// TIA Portal project "Tester_Forma_W1" (V16)
// Program sterowania formą wtryskarki do zalewania gumą końcuwek rur.

(* hardware
DEVICE "Tester_Forma"  S7-1200 Station
   slot 0: "Rack_0"  S7-1200 Rack  Rack  V1.0
   slot 1: "PLC_1"  CPU 1214C AC/DC/Rly  6ES7 214-1BG40-0XB0  V4.4
   slot 2: "DI 16x24VDC/DQ 16xRelay_1"  SM 1223 DI16/DQ16 x relay  6ES7 223-1PL32-0XB0  V2.0
   slot 3: "DQ 8x24VDC _1"  SM 1222 DQ8 x 24VDC  6ES7 222-1BF32-0XB0  V2.0
DEVICE "HMI_1"  KTP400 Basic PN
   slot 0: "HMI_1"  KTP400 Basic PN  6AV2 123-2DB03-0AX0  15.1.0.0
   slot 1: "HMI_RT_1"  KTP400 Basic PN  6AV2 123-2DB03-0AX0  15.1.0.0
   slot 5: "HMI_1.IE_CP_1"  PROFINET Interface  15.0.1.0
      slot 1: "PROFINET Interface_1"  PROFINET Interface
         slot 1: "Port_1"  Port
*)

// ===== PLC "PLC_1"  CPU 1214C AC/DC/Rly =====

VAR_GLOBAL   // PLC tag table "Default tag table"
   "System_Byte" AT %MB1 : Byte;
   "FirstScan" AT %M1.0 : Bool;
   "DiagStatusUpdate" AT %M1.1 : Bool;
   "AlwaysTRUE" AT %M1.2 : Bool;
   "AlwaysFALSE" AT %M1.3 : Bool;
   "Clock_Byte" AT %MB0 : Byte;
   "Clock_10Hz" AT %M0.0 : Bool;
   "Clock_5Hz" AT %M0.1 : Bool;
   "Clock_2.5Hz" AT %M0.2 : Bool;
   "Clock_2Hz" AT %M0.3 : Bool;
   "Clock_1.25Hz" AT %M0.4 : Bool;
   "Clock_1Hz" AT %M0.5 : Bool;
   "Clock_0.625Hz" AT %M0.6 : Bool;
   "Clock_0.5Hz" AT %M0.7 : Bool;
END_VAR

VAR_GLOBAL   // PLC tag table "InputsPLC"
   "diSE_OpenGripper1" AT %I0.0 : Bool;
   "diSE_OpenGripper2" AT %I0.1 : Bool;
   "diSE_OpenGripper3" AT %I0.2 : Bool;
   "diSE_OpenGripper4" AT %I0.3 : Bool;
   "diSE_OpenGripper5" AT %I0.4 : Bool;
   "diSE_OpenGripper6" AT %I0.5 : Bool;
   "diSE_OpenGripper7" AT %I0.6 : Bool;
   "diSE_OpenGripper8" AT %I0.7 : Bool;
   "diSE_PresencePin1" AT %I1.0 : Bool;
   "diSE_PresencePin2" AT %I1.1 : Bool;
   "diSE_PresencePin3" AT %I1.2 : Bool;
   "diSE_PresencePin4" AT %I1.3 : Bool;
   "diSE_PresencePin5" AT %I1.4 : Bool;
   "diSE_PresencePin6" AT %I1.5 : Bool;
   "diSE_PresencePin7" AT %I8.0 : Bool;
   "diSE_PresencePin8" AT %I8.1 : Bool;
   "diSE_LeftActuatorGrippersUpPosition" AT %I8.2 : Bool;
   "diSE_LeftActuatorGrippersDownPosition" AT %I8.3 : Bool;
   "diSE_LeftActuatorTablePinsDownPosition" AT %I8.4 : Bool;
   "diSE_LeftActuatorTablePinsUpPositon" AT %I8.5 : Bool;
   "diSE_RightActuatorTablePinsDownPositon" AT %I8.6 : Bool;
   "diSE_RightActuatorTablePinsUpPosition" AT %I8.7 : Bool;
   "diSE_RightActuatorGripperUpPosition" AT %I9.0 : Bool;
   "diSE_RightActuatorGripperDownPositon" AT %I9.1 : Bool;
   "diPressOpenedUp" AT %I9.4 : Bool;
   "diPressClosedDown" AT %I9.6 : Bool;
   "diPreventaOK" AT %I9.2 : Bool;
   "diBT_Reset" AT %I9.3 : Bool;
   "diBT_StartCycle2" AT %I9.5 : Bool;
   "diPressInjectionEnd" AT %I9.7 : Bool;
END_VAR

VAR_GLOBAL   // PLC tag table "OutputsPLC"
   "dqPermitToClosePress" AT %Q0.0 : Bool;
   "dqPressInterface1" AT %Q0.1 : Bool;
   "dqPressInterface2" AT %Q0.2 : Bool;
   "dqPressInterface3" AT %Q0.3 : Bool;
   "dqReserveQ0_4" AT %Q0.4 : Bool;
   "dqReserveQ0_5" AT %Q0.5 : Bool;
   "dqLED_RedFault" AT %Q0.6 : Bool;
   "dqBuzzer" AT %Q0.7 : Bool;
   "dqReserveQ1_0" AT %Q1.0 : Bool;
   "dqReserveQ1_1" AT %Q1.1 : Bool;
   "dqTablePinsUp" AT %Q8.0 : Bool;
   "dqTablePinsDown" AT %Q8.1 : Bool;
   "dqGrippresDown" AT %Q8.2 : Bool;
   "dqGrippersUp" AT %Q8.3 : Bool;
   "dqOpeningGripper1" AT %Q8.4 : Bool;
   "dqClosingGripper1" AT %Q8.5 : Bool;
   "dqOpeningGripper2" AT %Q8.6 : Bool;
   "dqClosingGripper2" AT %Q8.7 : Bool;
   "dqOpeningGripper3" AT %Q9.0 : Bool;
   "dqClosingGripper3" AT %Q9.1 : Bool;
   "dqOpeningGripper4" AT %Q9.2 : Bool;
   "dqClosingGripper4" AT %Q9.3 : Bool;
   "dqOpeningGripper5" AT %Q9.4 : Bool;
   "dqClosingGripper5" AT %Q9.5 : Bool;
   "dqOpeningGripper6" AT %Q9.6 : Bool;
   "dqClosingGripper6" AT %Q9.7 : Bool;
   "dqOpeningGripper7" AT %Q12.0 : Bool;
   "dqClosingGripper7" AT %Q12.1 : Bool;
   "dqOpeningGripper8" AT %Q12.2 : Bool;
   "dqClosingGripper8" AT %Q12.3 : Bool;
   "dqReserveq12_4" AT %Q12.4 : Bool;
   "dqReserveq12_5" AT %Q12.5 : Bool;
   "dqReserveq12_6" AT %Q12.6 : Bool;
   "dqReserveq12_7" AT %Q12.7 : Bool;
END_VAR

DATA_BLOCK "Variable"   // DB1
{ S7_Optimized_Access := 'TRUE' }
VERSION : 0.1
   VAR
      FirstScanDone : Bool;
      SetMachineInitialStatus : Bool;
   END_VAR
   VAR RETAIN
      M_EvTableGrippres : Bool;
      M_EvTablePins : Bool;
   END_VAR
   VAR
      OutBuzzerPinActivatedByTube1 : Bool;
      OutBuzzerPinActivatedByTube2 : Bool;
      OutBuzzerPinActivatedByTube3 : Bool;
      OutBuzzerPinActivatedByTube4 : Bool;
      OutBuzzerPinActivatedByTube5 : Bool;
      OutBuzzerPinActivatedByTube6 : Bool;
      OutBuzzerPinActivatedByTube7 : Bool;
      OutBuzzerPinActivatedByTube8 : Bool;
   END_VAR
   VAR RETAIN
      BuzzerDurationSignal : Time := T#100ms;
   END_VAR
   VAR
      SignalBuzzerPinPresent : Bool;
      M_PinsNotActivated : Bool;
      M_PinsActivated : Bool;
      M_GrippersOpened : Bool;
      M_GrippersClosed : Bool;
      M_PinsTableUpPosition : Bool;
      M_PinsTableDownPosition : Bool;
      M_GrippersTableUpPositon : Bool;
      M_GrippersTableDownPositon : Bool;
      M_EvGripperOutput1 : Bool;
      M_EvGripperOutput2 : Bool;
      M_EvGripperOutput3 : Bool;
      M_EvGripperOutput4 : Bool;
      M_EvGripperOutput5 : Bool;
      M_EvGripperOutput6 : Bool;
      M_EvGripperOutput7 : Bool;
      M_EvGripperOutput8 : Bool;
      M_ReadyForFirstCycle : Bool;
      M_PreparePositionForFirstStart : Bool;
      M_StartCycleButtons : Bool;
      M_EvGrippresInitial : Bool;
      M_EvTablePinsInitial : Bool := false;
      M_EvGripperOutputInitial : Bool;
      M_AutomaticModePermissionToCloseGrippers : Bool;
   END_VAR
BEGIN
END_DATA_BLOCK

DATA_BLOCK "HMI"   // DB8
{ S7_Optimized_Access := 'FALSE' }
VERSION : 0.1
   VAR
      Auto : Bool := false;
      Manu : Bool;
      OpenInAutoGripper1 : Bool;
      OpenInAutoGripper2 : Bool;
      OpenInAutoGripper3 : Bool;
      OpenInAutoGripper4 : Bool;
      OpenInAutoGripper5 : Bool;
      OpenInAutoGripper6 : Bool;
      OpenInAutoGripper7 : Bool;
      OpenInAutoGripper8 : Bool;
      OpenInManuGripper1 : Bool;
      OpenInManuGripper2 : Bool;
      OpenInManuGripper3 : Bool;
      OpenInManuGripper4 : Bool;
      OpenInManuGripper5 : Bool;
      OpenInManuGripper6 : Bool;
      OpenInManuGripper7 : Bool;
      OpenInManuGripper8 : Bool;
      CloseInManuGripper1 : Bool;
      CloseInManuGripper2 : Bool;
      CloseInManuGripper3 : Bool;
      CloseInManuGripper4 : Bool;
      CloseInManuGripper5 : Bool;
      CloseInManuGripper6 : Bool;
      CloseInManuGripper7 : Bool;
      CloseInManuGripper8 : Bool;
      TableGrippersUP : Bool;
      TableGripperDown : Bool;
      TablePinsUp : Bool;
      TablePinsDown : Bool;
      OpenManuAllGrippers : Bool;
   END_VAR
BEGIN
END_DATA_BLOCK

DATA_BLOCK "MemoryEdge"   // DB9
{ S7_Optimized_Access := 'TRUE' }
VERSION : 0.1
   VAR
      Memory1 : Bool;
      Memory2 : Bool;
      Memory3 : Bool;
      Memory4 : Bool;
      Memory5 : Bool;
      Memory6 : Bool;
      Memory7 : Bool;
      Memory8 : Bool;
      Memory9 : Bool;
      Memory10 : Bool;
      Memory11 : Bool;
      Memory12 : Bool;
      Memory13 : Bool;
      Memory14 : Bool;
   END_VAR
BEGIN
END_DATA_BLOCK

DATA_BLOCK "Outputs_DB"   // DB16
{ S7_Optimized_Access := 'TRUE' }
VERSION : 0.1
// stored: InstanceOfName Outputs
"Outputs"
BEGIN
END_DATA_BLOCK

DATA_BLOCK "AlarmsBlock"   // DB17
{ S7_Optimized_Access := 'FALSE' }
VERSION : 0.1
   VAR
      AlarmOccurred : Bool;
      AlarmLeftActuatorGrippers : Bool;
      AlarmRightActuatorGrippers : Bool;
      AlarmLeftActuatorPins : Bool;
      AlarmRightActuatorPins : Bool;
      M_AlarmGripper1 : Bool;
      M_AlarmGripper2 : Bool;
      M_AlarmGripper3 : Bool;
      M_AlarmGripper4 : Bool;
      M_AlarmGripper5 : Bool;
      M_AlarmGripper6 : Bool;
      M_AlarmGripper7 : Bool;
      M_AlarmGripper8 : Bool;
   END_VAR
BEGIN
END_DATA_BLOCK

// folder: GripperError

DATA_BLOCK "Gripper6_Error"   // DB6
{ S7_Optimized_Access := 'TRUE' }
VERSION : 0.1
// stored: InstanceOfName GripperError
"GripperError"
BEGIN
END_DATA_BLOCK

DATA_BLOCK "Gripper1_Error"   // DB7
{ S7_Optimized_Access := 'TRUE' }
VERSION : 0.1
// stored: InstanceOfName GripperError
"GripperError"
BEGIN
END_DATA_BLOCK

DATA_BLOCK "Gripper2_Error"   // DB10
{ S7_Optimized_Access := 'TRUE' }
VERSION : 0.1
// stored: InstanceOfName GripperError
"GripperError"
BEGIN
END_DATA_BLOCK

DATA_BLOCK "Gripper3_Error"   // DB11
{ S7_Optimized_Access := 'TRUE' }
VERSION : 0.1
// stored: InstanceOfName GripperError
"GripperError"
BEGIN
END_DATA_BLOCK

DATA_BLOCK "Gripper4_Error"   // DB12
{ S7_Optimized_Access := 'TRUE' }
VERSION : 0.1
// stored: InstanceOfName GripperError
"GripperError"
BEGIN
END_DATA_BLOCK

DATA_BLOCK "Gripper5_Error"   // DB13
{ S7_Optimized_Access := 'TRUE' }
VERSION : 0.1
// stored: InstanceOfName GripperError
"GripperError"
BEGIN
END_DATA_BLOCK

DATA_BLOCK "Gripper7_Error"   // DB14
{ S7_Optimized_Access := 'TRUE' }
VERSION : 0.1
// stored: InstanceOfName GripperError
"GripperError"
BEGIN
END_DATA_BLOCK

DATA_BLOCK "Gripper8_Error"   // DB15
{ S7_Optimized_Access := 'TRUE' }
VERSION : 0.1
// stored: InstanceOfName GripperError
"GripperError"
BEGIN
END_DATA_BLOCK

// folder: GripperOpenClose

DATA_BLOCK "GripperOpenCloseAutoManu_DB1"   // DB18
{ S7_Optimized_Access := 'TRUE' }
VERSION : 0.1
// stored: InstanceOfName GripperOpenCloseAutoManu
"GripperOpenCloseAutoManu"
BEGIN
END_DATA_BLOCK

DATA_BLOCK "GripperOpenCloseAutoManu_DB"   // DB19
{ S7_Optimized_Access := 'TRUE' }
VERSION : 0.1
// stored: InstanceOfName GripperOpenCloseAutoManu
"GripperOpenCloseAutoManu"
BEGIN
END_DATA_BLOCK

DATA_BLOCK "GripperOpenCloseAutoManu_DB_1"   // DB20
{ S7_Optimized_Access := 'TRUE' }
VERSION : 0.1
// stored: InstanceOfName GripperOpenCloseAutoManu
"GripperOpenCloseAutoManu"
BEGIN
END_DATA_BLOCK

DATA_BLOCK "GripperOpenCloseAutoManu_DB_2"   // DB21
{ S7_Optimized_Access := 'TRUE' }
VERSION : 0.1
// stored: InstanceOfName GripperOpenCloseAutoManu
"GripperOpenCloseAutoManu"
BEGIN
END_DATA_BLOCK

DATA_BLOCK "GripperOpenCloseAutoManu_DB_3"   // DB22
{ S7_Optimized_Access := 'TRUE' }
VERSION : 0.1
// stored: InstanceOfName GripperOpenCloseAutoManu
"GripperOpenCloseAutoManu"
BEGIN
END_DATA_BLOCK

DATA_BLOCK "GripperOpenCloseAutoManu_DB_4"   // DB23
{ S7_Optimized_Access := 'TRUE' }
VERSION : 0.1
// stored: InstanceOfName GripperOpenCloseAutoManu
"GripperOpenCloseAutoManu"
BEGIN
END_DATA_BLOCK

DATA_BLOCK "GripperOpenCloseAutoManu_DB_5"   // DB24
{ S7_Optimized_Access := 'TRUE' }
VERSION : 0.1
// stored: InstanceOfName GripperOpenCloseAutoManu
"GripperOpenCloseAutoManu"
BEGIN
END_DATA_BLOCK

DATA_BLOCK "GripperOpenCloseAutoManu_DB_6"   // DB25
{ S7_Optimized_Access := 'TRUE' }
VERSION : 0.1
// stored: InstanceOfName GripperOpenCloseAutoManu
"GripperOpenCloseAutoManu"
BEGIN
END_DATA_BLOCK

// folder: System blocks/Program resources

DATA_BLOCK "TimeToAlarmLeftActuatoGrippers"   // DB2
{ S7_Optimized_Access := 'TRUE' }
AUTHOR : Simatic
FAMILY : IEC
NAME : IEC_TMR
VERSION : 1.0
// stored: InstanceOfName IEC_TIMER
"IEC_TIMER"
BEGIN
END_DATA_BLOCK

DATA_BLOCK "TimeToAlarmRightActuatoGrippers"   // DB3
{ S7_Optimized_Access := 'TRUE' }
AUTHOR : Simatic
FAMILY : IEC
NAME : IEC_TMR
VERSION : 1.0
// stored: InstanceOfName IEC_TIMER
"IEC_TIMER"
BEGIN
END_DATA_BLOCK

DATA_BLOCK "TimeToAlarmLeftActuatoPins"   // DB4
{ S7_Optimized_Access := 'TRUE' }
AUTHOR : Simatic
FAMILY : IEC
NAME : IEC_TMR
VERSION : 1.0
// stored: InstanceOfName IEC_TIMER
"IEC_TIMER"
BEGIN
END_DATA_BLOCK

DATA_BLOCK "TimeToAlarmRightActuatorPins"   // DB5
{ S7_Optimized_Access := 'TRUE' }
AUTHOR : Simatic
FAMILY : IEC
NAME : IEC_TMR
VERSION : 1.0
// stored: InstanceOfName IEC_TIMER
"IEC_TIMER"
BEGIN
END_DATA_BLOCK

// folder: (top level)

FUNCTION_BLOCK "Outputs"   // FB2, LAD
{ S7_Optimized_Access := 'TRUE' }
VERSION : 0.1
   VAR
      ElectricValve_Grippers : "ElectricValve";
      ElectricValve_TablePins : "ElectricValve";
      ElectricValve_Gripper1 : "ElectricValve";
      ElectricValve_Gripper2 : "ElectricValve";
      ElectricValve_Gripper3 : "ElectricValve";
      ElectricValve_Gripper4 : "ElectricValve";
      ElectricValve_Gripper5 : "ElectricValve";
      ElectricValve_Gripper6 : "ElectricValve";
      ElectricValve_Gripper7 : "ElectricValve";
      ElectricValve_Gripper8 : "ElectricValve";
      Gripper1_Present_Signal : "Buzzer";
      Gripper2_Present_Signal : "Buzzer";
      Gripper3_Present_Signal : "Buzzer";
      Gripper4_Present_Signal : "Buzzer";
      Gripper5_Present_Signal : "Buzzer";
      Gripper6_Present_Signal : "Buzzer";
      Gripper7_Present_Signal : "Buzzer";
      Gripper8_Present_Signal : "Buzzer";
   END_VAR
BEGIN

REGION Network 1: Actuator of Grippers control.
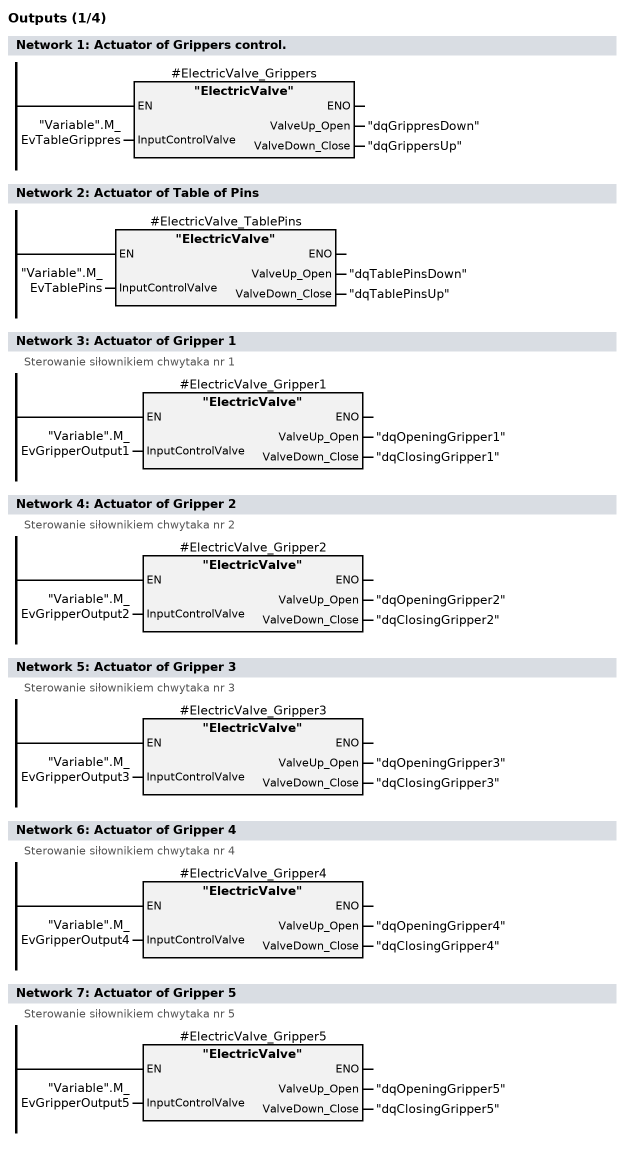
   RUNG wire#powerrail
      #ElectricValve_Grippers(InputControlValve := "Variable".M_EvTableGrippres, ValveUp_Open => "dqGrippresDown", ValveDown_Close => "dqGrippersUp")
   END_RUNG
   // the same network as SCL:
   #ElectricValve_Grippers(InputControlValve := "Variable".M_EvTableGrippres,   // "ElectricValve"
                           ValveUp_Open => "dqGrippresDown",
                           ValveDown_Close => "dqGrippersUp");
END_REGION

REGION Network 2: Actuator of Table of Pins
   RUNG wire#powerrail
      #ElectricValve_TablePins(InputControlValve := "Variable".M_EvTablePins, ValveUp_Open => "dqTablePinsDown", ValveDown_Close => "dqTablePinsUp")
   END_RUNG
   // the same network as SCL:
   #ElectricValve_TablePins(InputControlValve := "Variable".M_EvTablePins,   // "ElectricValve"
                           ValveUp_Open => "dqTablePinsDown",
                           ValveDown_Close => "dqTablePinsUp");
END_REGION

REGION Network 3: Actuator of Gripper 1
   // Sterowanie siłownikiem chwytaka nr 1
   RUNG wire#powerrail
      #ElectricValve_Gripper1(InputControlValve := "Variable".M_EvGripperOutput1, ValveUp_Open => "dqOpeningGripper1", ValveDown_Close => "dqClosingGripper1")
   END_RUNG
   // the same network as SCL:
   #ElectricValve_Gripper1(InputControlValve := "Variable".M_EvGripperOutput1,   // "ElectricValve"
                           ValveUp_Open => "dqOpeningGripper1",
                           ValveDown_Close => "dqClosingGripper1");
END_REGION

REGION Network 4: Actuator of Gripper 2
   // Sterowanie siłownikiem chwytaka nr 2
   RUNG wire#powerrail
      #ElectricValve_Gripper2(InputControlValve := "Variable".M_EvGripperOutput2, ValveUp_Open => "dqOpeningGripper2", ValveDown_Close => "dqClosingGripper2")
   END_RUNG
   // the same network as SCL:
   #ElectricValve_Gripper2(InputControlValve := "Variable".M_EvGripperOutput2,   // "ElectricValve"
                           ValveUp_Open => "dqOpeningGripper2",
                           ValveDown_Close => "dqClosingGripper2");
END_REGION

REGION Network 5: Actuator of Gripper 3
   // Sterowanie siłownikiem chwytaka nr 3
   RUNG wire#powerrail
      #ElectricValve_Gripper3(InputControlValve := "Variable".M_EvGripperOutput3, ValveUp_Open => "dqOpeningGripper3", ValveDown_Close => "dqClosingGripper3")
   END_RUNG
   // the same network as SCL:
   #ElectricValve_Gripper3(InputControlValve := "Variable".M_EvGripperOutput3,   // "ElectricValve"
                           ValveUp_Open => "dqOpeningGripper3",
                           ValveDown_Close => "dqClosingGripper3");
END_REGION

REGION Network 6: Actuator of Gripper 4
   // Sterowanie siłownikiem chwytaka nr 4
   RUNG wire#powerrail
      #ElectricValve_Gripper4(InputControlValve := "Variable".M_EvGripperOutput4, ValveUp_Open => "dqOpeningGripper4", ValveDown_Close => "dqClosingGripper4")
   END_RUNG
   // the same network as SCL:
   #ElectricValve_Gripper4(InputControlValve := "Variable".M_EvGripperOutput4,   // "ElectricValve"
                           ValveUp_Open => "dqOpeningGripper4",
                           ValveDown_Close => "dqClosingGripper4");
END_REGION

REGION Network 7: Actuator of Gripper 5
   // Sterowanie siłownikiem chwytaka nr 5
   RUNG wire#powerrail
      #ElectricValve_Gripper5(InputControlValve := "Variable".M_EvGripperOutput5, ValveUp_Open => "dqOpeningGripper5", ValveDown_Close => "dqClosingGripper5")
   END_RUNG
   // the same network as SCL:
   #ElectricValve_Gripper5(InputControlValve := "Variable".M_EvGripperOutput5,   // "ElectricValve"
                           ValveUp_Open => "dqOpeningGripper5",
                           ValveDown_Close => "dqClosingGripper5");
END_REGION

REGION Network 8: Actuator of Gripper 6
   // Sterowanie siłownikiem chwytaka nr  6
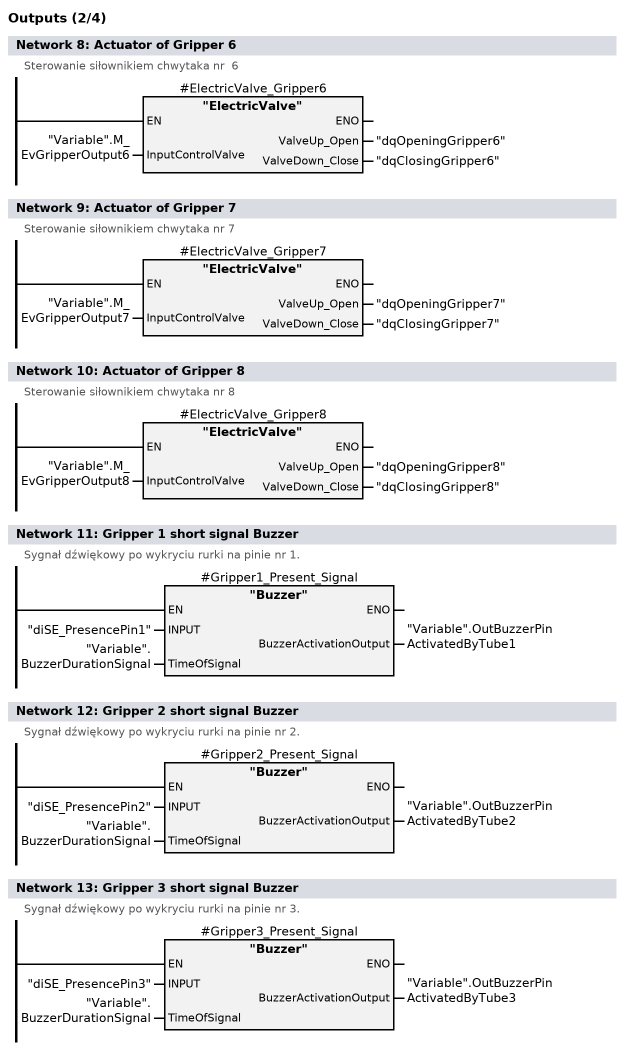
   RUNG wire#powerrail
      #ElectricValve_Gripper6(InputControlValve := "Variable".M_EvGripperOutput6, ValveUp_Open => "dqOpeningGripper6", ValveDown_Close => "dqClosingGripper6")
   END_RUNG
   // the same network as SCL:
   #ElectricValve_Gripper6(InputControlValve := "Variable".M_EvGripperOutput6,   // "ElectricValve"
                           ValveUp_Open => "dqOpeningGripper6",
                           ValveDown_Close => "dqClosingGripper6");
END_REGION

REGION Network 9: Actuator of Gripper 7
   // Sterowanie siłownikiem chwytaka nr 7
   RUNG wire#powerrail
      #ElectricValve_Gripper7(InputControlValve := "Variable".M_EvGripperOutput7, ValveUp_Open => "dqOpeningGripper7", ValveDown_Close => "dqClosingGripper7")
   END_RUNG
   // the same network as SCL:
   #ElectricValve_Gripper7(InputControlValve := "Variable".M_EvGripperOutput7,   // "ElectricValve"
                           ValveUp_Open => "dqOpeningGripper7",
                           ValveDown_Close => "dqClosingGripper7");
END_REGION

REGION Network 10: Actuator of Gripper 8
   // Sterowanie siłownikiem chwytaka nr 8
   RUNG wire#powerrail
      #ElectricValve_Gripper8(InputControlValve := "Variable".M_EvGripperOutput8, ValveUp_Open => "dqOpeningGripper8", ValveDown_Close => "dqClosingGripper8")
   END_RUNG
   // the same network as SCL:
   #ElectricValve_Gripper8(InputControlValve := "Variable".M_EvGripperOutput8,   // "ElectricValve"
                           ValveUp_Open => "dqOpeningGripper8",
                           ValveDown_Close => "dqClosingGripper8");
END_REGION

REGION Network 11: Gripper 1 short signal Buzzer
   // Sygnał dźwiękowy po wykryciu rurki na pinie nr 1.
   RUNG wire#powerrail
      #Gripper1_Present_Signal(INPUT := "diSE_PresencePin1", TimeOfSignal := "Variable".BuzzerDurationSignal, BuzzerActivationOutput => "Variable".OutBuzzerPinActivatedByTube1)
   END_RUNG
   // the same network as SCL:
   #Gripper1_Present_Signal(INPUT := "diSE_PresencePin1",   // "Buzzer"
                           TimeOfSignal := "Variable".BuzzerDurationSignal,
                           BuzzerActivationOutput => "Variable".OutBuzzerPinActivatedByTube1);
END_REGION

REGION Network 12: Gripper 2 short signal Buzzer
   // Sygnał dźwiękowy po wykryciu rurki na pinie nr 2.
   RUNG wire#powerrail
      #Gripper2_Present_Signal(INPUT := "diSE_PresencePin2", TimeOfSignal := "Variable".BuzzerDurationSignal, BuzzerActivationOutput => "Variable".OutBuzzerPinActivatedByTube2)
   END_RUNG
   // the same network as SCL:
   #Gripper2_Present_Signal(INPUT := "diSE_PresencePin2",   // "Buzzer"
                           TimeOfSignal := "Variable".BuzzerDurationSignal,
                           BuzzerActivationOutput => "Variable".OutBuzzerPinActivatedByTube2);
END_REGION

REGION Network 13: Gripper 3 short signal Buzzer
   // Sygnał dźwiękowy po wykryciu rurki na pinie nr 3.
   RUNG wire#powerrail
      #Gripper3_Present_Signal(INPUT := "diSE_PresencePin3", TimeOfSignal := "Variable".BuzzerDurationSignal, BuzzerActivationOutput => "Variable".OutBuzzerPinActivatedByTube3)
   END_RUNG
   // the same network as SCL:
   #Gripper3_Present_Signal(INPUT := "diSE_PresencePin3",   // "Buzzer"
                           TimeOfSignal := "Variable".BuzzerDurationSignal,
                           BuzzerActivationOutput => "Variable".OutBuzzerPinActivatedByTube3);
END_REGION

REGION Network 14: Gripper 4 short signal Buzzer
   // Sygnał dźwiękowy po wykryciu rurki na pinie nr 4.
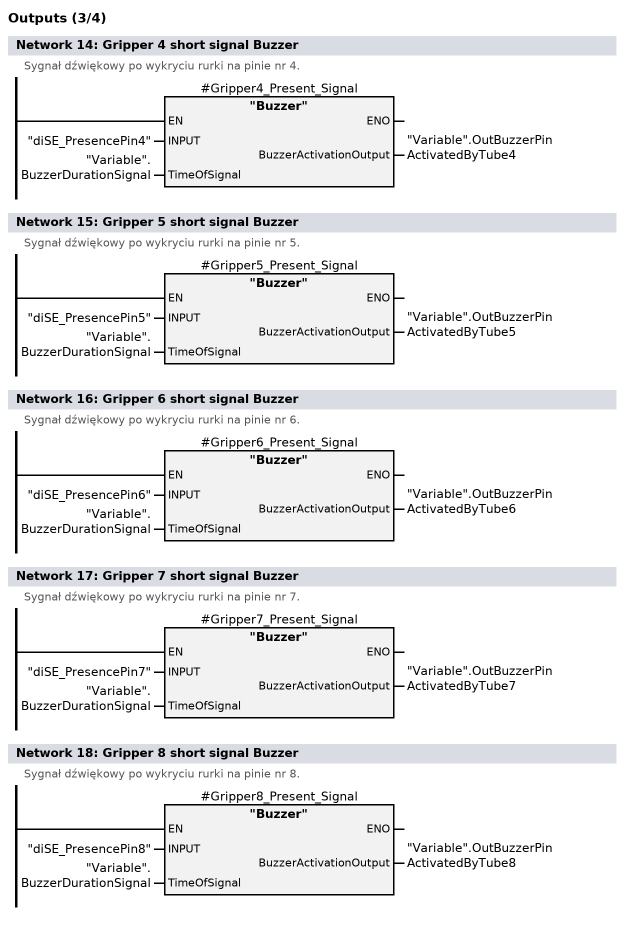
   RUNG wire#powerrail
      #Gripper4_Present_Signal(INPUT := "diSE_PresencePin4", TimeOfSignal := "Variable".BuzzerDurationSignal, BuzzerActivationOutput => "Variable".OutBuzzerPinActivatedByTube4)
   END_RUNG
   // the same network as SCL:
   #Gripper4_Present_Signal(INPUT := "diSE_PresencePin4",   // "Buzzer"
                           TimeOfSignal := "Variable".BuzzerDurationSignal,
                           BuzzerActivationOutput => "Variable".OutBuzzerPinActivatedByTube4);
END_REGION

REGION Network 15: Gripper 5 short signal Buzzer
   // Sygnał dźwiękowy po wykryciu rurki na pinie nr 5.
   RUNG wire#powerrail
      #Gripper5_Present_Signal(INPUT := "diSE_PresencePin5", TimeOfSignal := "Variable".BuzzerDurationSignal, BuzzerActivationOutput => "Variable".OutBuzzerPinActivatedByTube5)
   END_RUNG
   // the same network as SCL:
   #Gripper5_Present_Signal(INPUT := "diSE_PresencePin5",   // "Buzzer"
                           TimeOfSignal := "Variable".BuzzerDurationSignal,
                           BuzzerActivationOutput => "Variable".OutBuzzerPinActivatedByTube5);
END_REGION

REGION Network 16: Gripper 6 short signal Buzzer
   // Sygnał dźwiękowy po wykryciu rurki na pinie nr 6.
   RUNG wire#powerrail
      #Gripper6_Present_Signal(INPUT := "diSE_PresencePin6", TimeOfSignal := "Variable".BuzzerDurationSignal, BuzzerActivationOutput => "Variable".OutBuzzerPinActivatedByTube6)
   END_RUNG
   // the same network as SCL:
   #Gripper6_Present_Signal(INPUT := "diSE_PresencePin6",   // "Buzzer"
                           TimeOfSignal := "Variable".BuzzerDurationSignal,
                           BuzzerActivationOutput => "Variable".OutBuzzerPinActivatedByTube6);
END_REGION

REGION Network 17: Gripper 7 short signal Buzzer
   // Sygnał dźwiękowy po wykryciu rurki na pinie nr 7.
   RUNG wire#powerrail
      #Gripper7_Present_Signal(INPUT := "diSE_PresencePin7", TimeOfSignal := "Variable".BuzzerDurationSignal, BuzzerActivationOutput => "Variable".OutBuzzerPinActivatedByTube7)
   END_RUNG
   // the same network as SCL:
   #Gripper7_Present_Signal(INPUT := "diSE_PresencePin7",   // "Buzzer"
                           TimeOfSignal := "Variable".BuzzerDurationSignal,
                           BuzzerActivationOutput => "Variable".OutBuzzerPinActivatedByTube7);
END_REGION

REGION Network 18: Gripper 8 short signal Buzzer
   // Sygnał dźwiękowy po wykryciu rurki na pinie nr 8.
   RUNG wire#powerrail
      #Gripper8_Present_Signal(INPUT := "diSE_PresencePin8", TimeOfSignal := "Variable".BuzzerDurationSignal, BuzzerActivationOutput => "Variable".OutBuzzerPinActivatedByTube8)
   END_RUNG
   // the same network as SCL:
   #Gripper8_Present_Signal(INPUT := "diSE_PresencePin8",   // "Buzzer"
                           TimeOfSignal := "Variable".BuzzerDurationSignal,
                           BuzzerActivationOutput => "Variable".OutBuzzerPinActivatedByTube8);
END_REGION

REGION Network 19: Signal of Buzzer after pin activation
   // Sygnał dźwiękowy po aktywacji jednego z pinów.
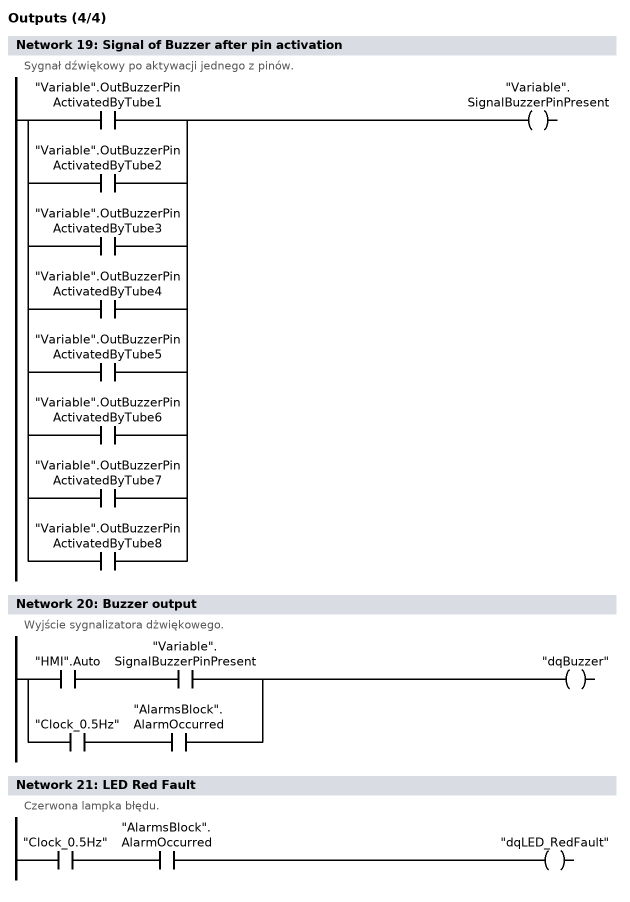
   RUNG wire#powerrail
      Contact( "Variable".OutBuzzerPinActivatedByTube1 )
      wire#w1
      Coil( "Variable".SignalBuzzerPinPresent )
   END_RUNG
   RUNG wire#powerrail
      Contact( "Variable".OutBuzzerPinActivatedByTube2 )
   END_RUNG wire#w1
   RUNG wire#powerrail
      Contact( "Variable".OutBuzzerPinActivatedByTube3 )
   END_RUNG wire#w1
   RUNG wire#powerrail
      Contact( "Variable".OutBuzzerPinActivatedByTube4 )
   END_RUNG wire#w1
   RUNG wire#powerrail
      Contact( "Variable".OutBuzzerPinActivatedByTube5 )
   END_RUNG wire#w1
   RUNG wire#powerrail
      Contact( "Variable".OutBuzzerPinActivatedByTube6 )
   END_RUNG wire#w1
   RUNG wire#powerrail
      Contact( "Variable".OutBuzzerPinActivatedByTube7 )
   END_RUNG wire#w1
   RUNG wire#powerrail
      Contact( "Variable".OutBuzzerPinActivatedByTube8 )
   END_RUNG wire#w1
   // the same network as SCL:
   "Variable".SignalBuzzerPinPresent := "Variable".OutBuzzerPinActivatedByTube1 OR "Variable".OutBuzzerPinActivatedByTube2 OR "Variable".OutBuzzerPinActivatedByTube3 OR "Variable".OutBuzzerPinActivatedByTube4 OR "Variable".OutBuzzerPinActivatedByTube5 OR "Variable".OutBuzzerPinActivatedByTube6 OR "Variable".OutBuzzerPinActivatedByTube7 OR "Variable".OutBuzzerPinActivatedByTube8;
END_REGION

REGION Network 20: Buzzer output
   // Wyjście sygnalizatora dżwiękowego.
   RUNG wire#powerrail
      Contact( "HMI".Auto )
      Contact( "Variable".SignalBuzzerPinPresent )
      wire#w1
      Coil( "dqBuzzer" )
   END_RUNG
   RUNG wire#powerrail
      Contact( "Clock_0.5Hz" )
      Contact( "AlarmsBlock".AlarmOccurred )
   END_RUNG wire#w1
   // the same network as SCL:
   "dqBuzzer" := ("HMI".Auto AND "Variable".SignalBuzzerPinPresent) OR ("Clock_0.5Hz" AND "AlarmsBlock".AlarmOccurred);
END_REGION

REGION Network 21: LED Red Fault
   // Czerwona lampka błędu.
   RUNG wire#powerrail
      Contact( "Clock_0.5Hz" )
      Contact( "AlarmsBlock".AlarmOccurred )
      Coil( "dqLED_RedFault" )
   END_RUNG
   // the same network as SCL:
   "dqLED_RedFault" := "Clock_0.5Hz" AND "AlarmsBlock".AlarmOccurred;
END_REGION
END_FUNCTION_BLOCK

FUNCTION "Cycle" : Void   // FC1, LAD
{ S7_Optimized_Access := 'TRUE' }
VERSION : 0.1
   VAR_TEMP   // added for the SCL form of the ladder/FBD networks
      _w1 : Bool;
   END_VAR
BEGIN

REGION Network 1: Checking the starting position of the machine - pins are activated or not activated
   // Sprawdzenie, czy czujniki pinów sa aktywne.
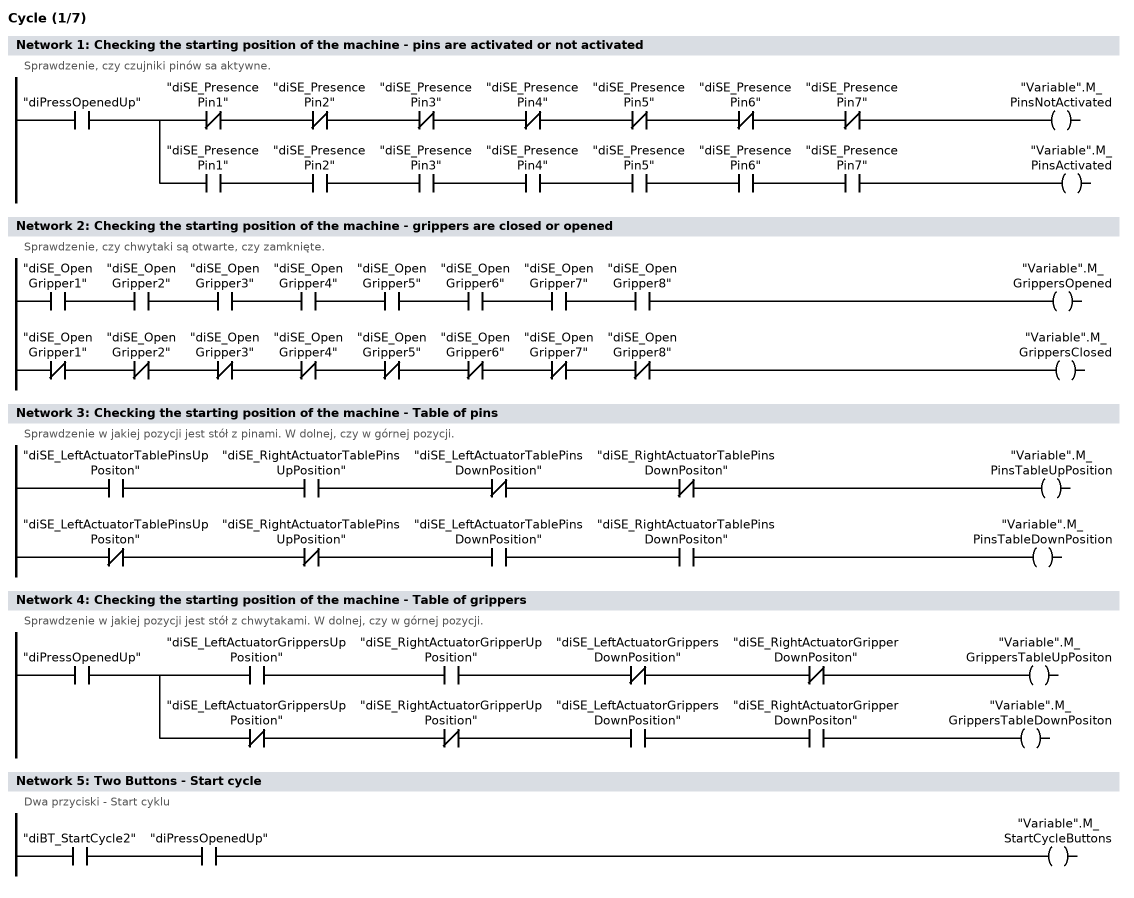
   RUNG wire#powerrail
      Contact( "diPressOpenedUp" )
      wire#w1
      I_Contact( "diSE_PresencePin1" )
      I_Contact( "diSE_PresencePin2" )
      I_Contact( "diSE_PresencePin3" )
      I_Contact( "diSE_PresencePin4" )
      I_Contact( "diSE_PresencePin5" )
      I_Contact( "diSE_PresencePin6" )
      I_Contact( "diSE_PresencePin7" )
      Coil( "Variable".M_PinsNotActivated )
   END_RUNG
   RUNG wire#w1
      Contact( "diSE_PresencePin1" )
      Contact( "diSE_PresencePin2" )
      Contact( "diSE_PresencePin3" )
      Contact( "diSE_PresencePin4" )
      Contact( "diSE_PresencePin5" )
      Contact( "diSE_PresencePin6" )
      Contact( "diSE_PresencePin7" )
      Coil( "Variable".M_PinsActivated )
   END_RUNG
   // the same network as SCL:
   "Variable".M_PinsNotActivated := "diPressOpenedUp" AND NOT "diSE_PresencePin1" AND NOT "diSE_PresencePin2" AND NOT "diSE_PresencePin3" AND NOT "diSE_PresencePin4" AND NOT "diSE_PresencePin5" AND NOT "diSE_PresencePin6" AND NOT "diSE_PresencePin7";
   "Variable".M_PinsActivated := "diPressOpenedUp" AND "diSE_PresencePin1" AND "diSE_PresencePin2" AND "diSE_PresencePin3" AND "diSE_PresencePin4" AND "diSE_PresencePin5" AND "diSE_PresencePin6" AND "diSE_PresencePin7";
END_REGION

REGION Network 2: Checking the starting position of the machine - grippers are closed or opened
   // Sprawdzenie, czy chwytaki są otwarte, czy zamknięte.
   RUNG wire#powerrail
      Contact( "diSE_OpenGripper1" )
      Contact( "diSE_OpenGripper2" )
      Contact( "diSE_OpenGripper3" )
      Contact( "diSE_OpenGripper4" )
      Contact( "diSE_OpenGripper5" )
      Contact( "diSE_OpenGripper6" )
      Contact( "diSE_OpenGripper7" )
      Contact( "diSE_OpenGripper8" )
      Coil( "Variable".M_GrippersOpened )
   END_RUNG
   RUNG wire#powerrail
      I_Contact( "diSE_OpenGripper1" )
      I_Contact( "diSE_OpenGripper2" )
      I_Contact( "diSE_OpenGripper3" )
      I_Contact( "diSE_OpenGripper4" )
      I_Contact( "diSE_OpenGripper5" )
      I_Contact( "diSE_OpenGripper6" )
      I_Contact( "diSE_OpenGripper7" )
      I_Contact( "diSE_OpenGripper8" )
      Coil( "Variable".M_GrippersClosed )
   END_RUNG
   // the same network as SCL:
   "Variable".M_GrippersOpened := "diSE_OpenGripper1" AND "diSE_OpenGripper2" AND "diSE_OpenGripper3" AND "diSE_OpenGripper4" AND "diSE_OpenGripper5" AND "diSE_OpenGripper6" AND "diSE_OpenGripper7" AND "diSE_OpenGripper8";
   "Variable".M_GrippersClosed := NOT "diSE_OpenGripper1" AND NOT "diSE_OpenGripper2" AND NOT "diSE_OpenGripper3" AND NOT "diSE_OpenGripper4" AND NOT "diSE_OpenGripper5" AND NOT "diSE_OpenGripper6" AND NOT "diSE_OpenGripper7" AND NOT "diSE_OpenGripper8";
END_REGION

REGION Network 3: Checking the starting position of the machine - Table of pins
   // Sprawdzenie w jakiej pozycji jest stół z pinami. W dolnej, czy w górnej pozycji.
   RUNG wire#powerrail
      Contact( "diSE_LeftActuatorTablePinsUpPositon" )
      Contact( "diSE_RightActuatorTablePinsUpPosition" )
      I_Contact( "diSE_LeftActuatorTablePinsDownPosition" )
      I_Contact( "diSE_RightActuatorTablePinsDownPositon" )
      Coil( "Variable".M_PinsTableUpPosition )
   END_RUNG
   RUNG wire#powerrail
      I_Contact( "diSE_LeftActuatorTablePinsUpPositon" )
      I_Contact( "diSE_RightActuatorTablePinsUpPosition" )
      Contact( "diSE_LeftActuatorTablePinsDownPosition" )
      Contact( "diSE_RightActuatorTablePinsDownPositon" )
      Coil( "Variable".M_PinsTableDownPosition )
   END_RUNG
   // the same network as SCL:
   "Variable".M_PinsTableUpPosition := "diSE_LeftActuatorTablePinsUpPositon" AND "diSE_RightActuatorTablePinsUpPosition" AND NOT "diSE_LeftActuatorTablePinsDownPosition" AND NOT "diSE_RightActuatorTablePinsDownPositon";
   "Variable".M_PinsTableDownPosition := NOT "diSE_LeftActuatorTablePinsUpPositon" AND NOT "diSE_RightActuatorTablePinsUpPosition" AND "diSE_LeftActuatorTablePinsDownPosition" AND "diSE_RightActuatorTablePinsDownPositon";
END_REGION

REGION Network 4: Checking the starting position of the machine - Table of grippers
   // Sprawdzenie w jakiej pozycji jest stół z chwytakami. W dolnej, czy w górnej pozycji.
   RUNG wire#powerrail
      Contact( "diPressOpenedUp" )
      wire#w1
      Contact( "diSE_LeftActuatorGrippersUpPosition" )
      Contact( "diSE_RightActuatorGripperUpPosition" )
      I_Contact( "diSE_LeftActuatorGrippersDownPosition" )
      I_Contact( "diSE_RightActuatorGripperDownPositon" )
      Coil( "Variable".M_GrippersTableUpPositon )
   END_RUNG
   RUNG wire#w1
      I_Contact( "diSE_LeftActuatorGrippersUpPosition" )
      I_Contact( "diSE_RightActuatorGripperUpPosition" )
      Contact( "diSE_LeftActuatorGrippersDownPosition" )
      Contact( "diSE_RightActuatorGripperDownPositon" )
      Coil( "Variable".M_GrippersTableDownPositon )
   END_RUNG
   // the same network as SCL:
   "Variable".M_GrippersTableUpPositon := "diPressOpenedUp" AND "diSE_LeftActuatorGrippersUpPosition" AND "diSE_RightActuatorGripperUpPosition" AND NOT "diSE_LeftActuatorGrippersDownPosition" AND NOT "diSE_RightActuatorGripperDownPositon";
   "Variable".M_GrippersTableDownPositon := "diPressOpenedUp" AND NOT "diSE_LeftActuatorGrippersUpPosition" AND NOT "diSE_RightActuatorGripperUpPosition" AND "diSE_LeftActuatorGrippersDownPosition" AND "diSE_RightActuatorGripperDownPositon";
END_REGION

REGION Network 5: Two Buttons - Start cycle
   // Dwa przyciski - Start cyklu
   RUNG wire#powerrail
      Contact( "diBT_StartCycle2" )
      Contact( "diPressOpenedUp" )
      Coil( "Variable".M_StartCycleButtons )
   END_RUNG
   // the same network as SCL:
   "Variable".M_StartCycleButtons := "diBT_StartCycle2" AND "diPressOpenedUp";
END_REGION

REGION Network 6: Electrovalve of Table Gripper Control
   // Sterownaie elektrozaworem podnoszenia i opuszczania stołu chwytaków. Stół chwytaków jest w pozycji górnej, gdy zmiennna
   // "Variable".M_EvTableGrippres = 1. Gdy równa się 0, stół chwytaków jest w pozycji dolnej.
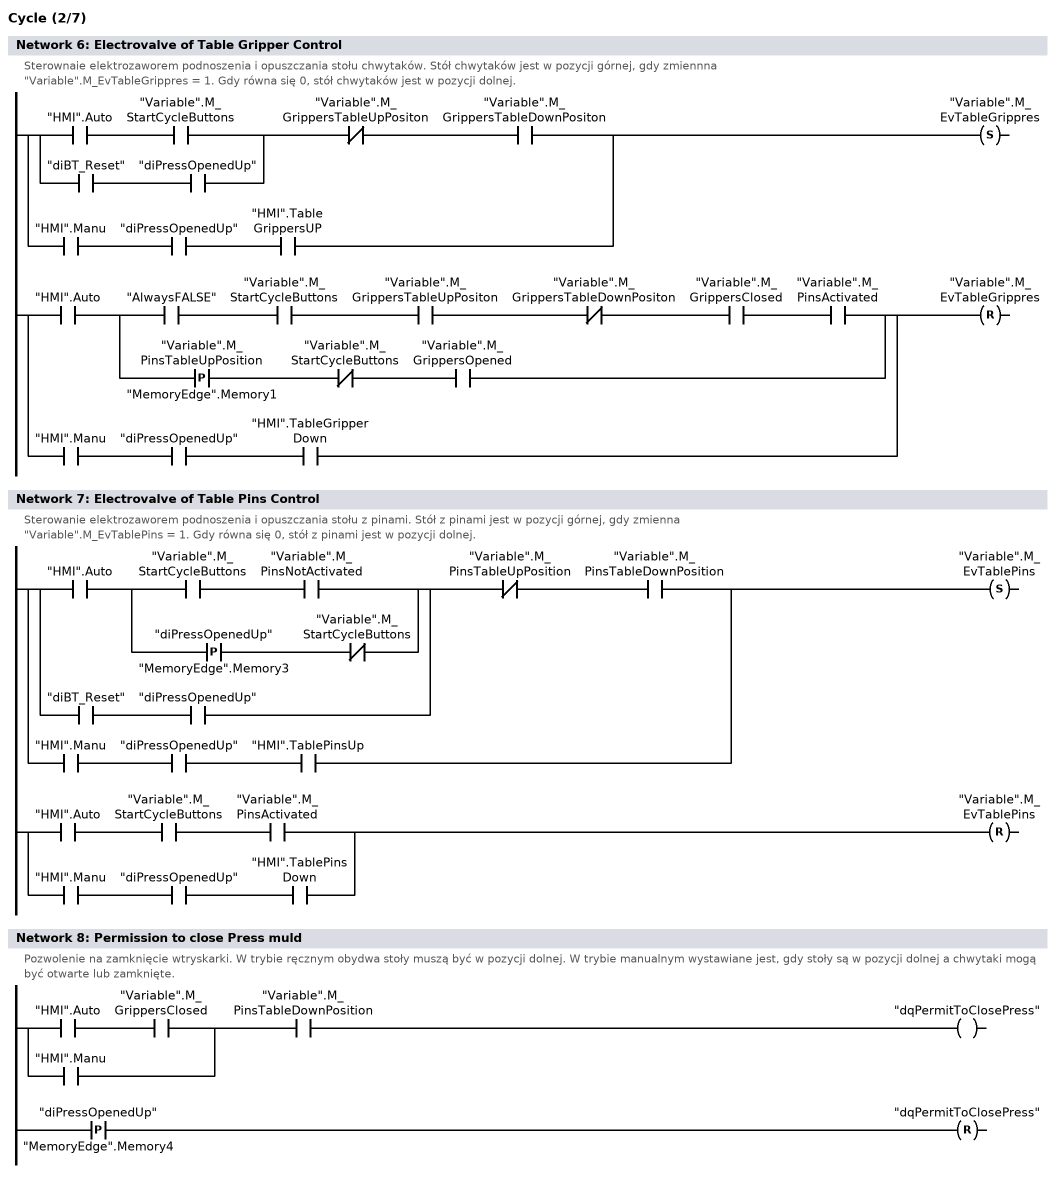
   RUNG wire#powerrail
      Contact( "HMI".Auto )
      Contact( "Variable".M_StartCycleButtons )
      wire#w1
      I_Contact( "Variable".M_GrippersTableUpPositon )
      Contact( "Variable".M_GrippersTableDownPositon )
      wire#w2
      S_Coil( "Variable".M_EvTableGrippres )
   END_RUNG
   RUNG wire#powerrail
      Contact( "diBT_Reset" )
      Contact( "diPressOpenedUp" )
   END_RUNG wire#w1
   RUNG wire#powerrail
      Contact( "HMI".Manu )
      Contact( "diPressOpenedUp" )
      Contact( "HMI".TableGrippersUP )
   END_RUNG wire#w2
   RUNG wire#powerrail
      Contact( "HMI".Auto )
      wire#w3
      Contact( "AlwaysFALSE" )
      Contact( "Variable".M_StartCycleButtons )
      Contact( "Variable".M_GrippersTableUpPositon )
      I_Contact( "Variable".M_GrippersTableDownPositon )
      Contact( "Variable".M_GrippersClosed )
      Contact( "Variable".M_PinsActivated )
      wire#w4
      R_Coil( "Variable".M_EvTableGrippres )
   END_RUNG
   RUNG wire#w3
      P_Contact(operand := "Variable".M_PinsTableUpPosition, bit := "MemoryEdge".Memory1)
      I_Contact( "Variable".M_StartCycleButtons )
      Contact( "Variable".M_GrippersOpened )
   END_RUNG wire#w4
   RUNG wire#powerrail
      Contact( "HMI".Manu )
      Contact( "diPressOpenedUp" )
      Contact( "HMI".TableGripperDown )
   END_RUNG wire#w4
   // the same network as SCL:
   IF ((("HMI".Auto AND "Variable".M_StartCycleButtons) OR ("diBT_Reset" AND "diPressOpenedUp")) AND NOT "Variable".M_GrippersTableUpPositon AND "Variable".M_GrippersTableDownPositon) OR ("HMI".Manu AND "diPressOpenedUp" AND "HMI".TableGrippersUP) THEN
       "Variable".M_EvTableGrippres := TRUE;
   END_IF;
   #_w1 := "HMI".Auto AND "Variable".M_PinsTableUpPosition AND NOT "MemoryEdge".Memory1;   // rising edge of "Variable".M_PinsTableUpPosition
   "MemoryEdge".Memory1 := "Variable".M_PinsTableUpPosition;
   IF ("HMI".Auto AND "AlwaysFALSE" AND "Variable".M_StartCycleButtons AND "Variable".M_GrippersTableUpPositon AND NOT "Variable".M_GrippersTableDownPositon AND "Variable".M_GrippersClosed AND "Variable".M_PinsActivated) OR (#_w1 AND NOT "Variable".M_StartCycleButtons AND "Variable".M_GrippersOpened) OR ("HMI".Manu AND "diPressOpenedUp" AND "HMI".TableGripperDown) THEN
       "Variable".M_EvTableGrippres := FALSE;
   END_IF;
END_REGION

REGION Network 7: Electrovalve of Table Pins Control
   // Sterowanie elektrozaworem podnoszenia i opuszczania stołu z pinami. Stół z pinami jest w pozycji górnej, gdy zmienna
   // "Variable".M_EvTablePins = 1. Gdy równa się 0, stół z pinami jest w pozycji dolnej.
   RUNG wire#powerrail
      Contact( "HMI".Auto )
      wire#w1
      Contact( "Variable".M_StartCycleButtons )
      Contact( "Variable".M_PinsNotActivated )
      wire#w2
      I_Contact( "Variable".M_PinsTableUpPosition )
      Contact( "Variable".M_PinsTableDownPosition )
      wire#w3
      S_Coil( "Variable".M_EvTablePins )
   END_RUNG
   RUNG wire#w1
      P_Contact(operand := "diPressOpenedUp", bit := "MemoryEdge".Memory3)
      I_Contact( "Variable".M_StartCycleButtons )
   END_RUNG wire#w2
   RUNG wire#powerrail
      Contact( "diBT_Reset" )
      Contact( "diPressOpenedUp" )
   END_RUNG wire#w2
   RUNG wire#powerrail
      Contact( "HMI".Manu )
      Contact( "diPressOpenedUp" )
      Contact( "HMI".TablePinsUp )
   END_RUNG wire#w3
   RUNG wire#powerrail
      Contact( "HMI".Auto )
      Contact( "Variable".M_StartCycleButtons )
      Contact( "Variable".M_PinsActivated )
      wire#w4
      R_Coil( "Variable".M_EvTablePins )
   END_RUNG
   RUNG wire#powerrail
      Contact( "HMI".Manu )
      Contact( "diPressOpenedUp" )
      Contact( "HMI".TablePinsDown )
   END_RUNG wire#w4
   // the same network as SCL:
   #_w1 := "HMI".Auto AND "diPressOpenedUp" AND NOT "MemoryEdge".Memory3;   // rising edge of "diPressOpenedUp"
   "MemoryEdge".Memory3 := "diPressOpenedUp";
   IF ((("HMI".Auto AND "Variable".M_StartCycleButtons AND "Variable".M_PinsNotActivated) OR (#_w1 AND NOT "Variable".M_StartCycleButtons) OR ("diBT_Reset" AND "diPressOpenedUp")) AND NOT "Variable".M_PinsTableUpPosition AND "Variable".M_PinsTableDownPosition) OR ("HMI".Manu AND "diPressOpenedUp" AND "HMI".TablePinsUp) THEN
       "Variable".M_EvTablePins := TRUE;
   END_IF;
   IF ("HMI".Auto AND "Variable".M_StartCycleButtons AND "Variable".M_PinsActivated) OR ("HMI".Manu AND "diPressOpenedUp" AND "HMI".TablePinsDown) THEN
       "Variable".M_EvTablePins := FALSE;
   END_IF;
END_REGION

REGION Network 8: Permission to close Press muld
   // Pozwolenie na zamknięcie wtryskarki. W trybie ręcznym obydwa stoły muszą być w pozycji dolnej. W trybie manualnym wystawiane jest, gdy stoły są w pozycji dolnej a chwytaki mogą być otwarte lub zamknięte.
   RUNG wire#powerrail
      Contact( "HMI".Auto )
      Contact( "Variable".M_GrippersClosed )
      wire#w1
      Contact( "Variable".M_PinsTableDownPosition )
      Coil( "dqPermitToClosePress" )
   END_RUNG
   RUNG wire#powerrail
      Contact( "HMI".Manu )
   END_RUNG wire#w1
   RUNG wire#powerrail
      P_Contact(operand := "diPressOpenedUp", bit := "MemoryEdge".Memory4)
      R_Coil( "dqPermitToClosePress" )
   END_RUNG
   // the same network as SCL:
   "dqPermitToClosePress" := (("HMI".Auto AND "Variable".M_GrippersClosed) OR "HMI".Manu) AND "Variable".M_PinsTableDownPosition;
   #_w1 := "diPressOpenedUp" AND NOT "MemoryEdge".Memory4;   // rising edge of "diPressOpenedUp"
   "MemoryEdge".Memory4 := "diPressOpenedUp";
   IF #_w1 THEN "dqPermitToClosePress" := FALSE; END_IF;
END_REGION

REGION Network 9: Permission for close the grippers in Automatic mode
   // Pozwolenie na zamykanie chwytaków w trybie automatycznym. Stół z chwytakami i stół z pinami są w górnych pozycjach.
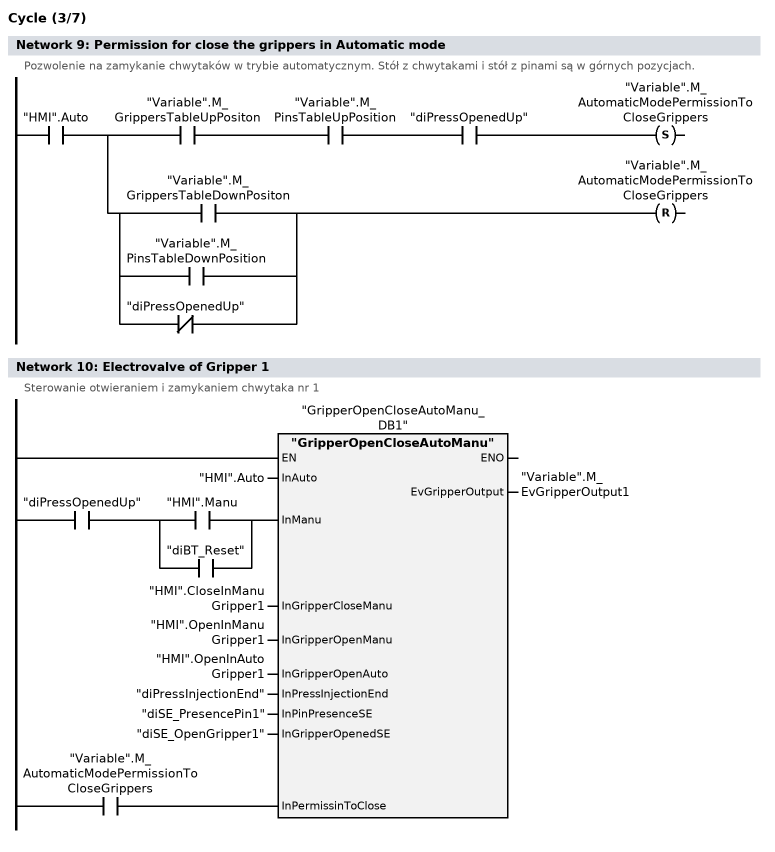
   RUNG wire#powerrail
      Contact( "HMI".Auto )
      wire#w1
      Contact( "Variable".M_GrippersTableUpPositon )
      Contact( "Variable".M_PinsTableUpPosition )
      Contact( "diPressOpenedUp" )
      S_Coil( "Variable".M_AutomaticModePermissionToCloseGrippers )
   END_RUNG
   RUNG wire#w1
      Contact( "Variable".M_GrippersTableDownPositon )
      wire#w2
      R_Coil( "Variable".M_AutomaticModePermissionToCloseGrippers )
   END_RUNG
   RUNG wire#w1
      Contact( "Variable".M_PinsTableDownPosition )
   END_RUNG wire#w2
   RUNG wire#w1
      I_Contact( "diPressOpenedUp" )
   END_RUNG wire#w2
   // the same network as SCL:
   IF "HMI".Auto AND "Variable".M_GrippersTableUpPositon AND "Variable".M_PinsTableUpPosition AND "diPressOpenedUp" THEN
       "Variable".M_AutomaticModePermissionToCloseGrippers := TRUE;
   END_IF;
   IF "HMI".Auto AND ("Variable".M_GrippersTableDownPositon OR "Variable".M_PinsTableDownPosition OR NOT "diPressOpenedUp") THEN
       "Variable".M_AutomaticModePermissionToCloseGrippers := FALSE;
   END_IF;
END_REGION

REGION Network 10: Electrovalve of Gripper 1
   // Sterowanie otwieraniem i zamykaniem chwytaka nr 1
   RUNG wire#powerrail
      "GripperOpenCloseAutoManu_DB1"(InManu := wire#w2, InPermissinToClose := wire#w3, InAuto := "HMI".Auto, InGripperCloseManu := "HMI".CloseInManuGripper1, InGripperOpenManu := "HMI".OpenInManuGripper1, InGripperOpenAuto := "HMI".OpenInAutoGripper1, InPressInjectionEnd := "diPressInjectionEnd", InPinPresenceSE := "diSE_PresencePin1", InGripperOpenedSE := "diSE_OpenGripper1", EvGripperOutput => "Variable".M_EvGripperOutput1)
   END_RUNG
   RUNG wire#powerrail
      Contact( "diPressOpenedUp" )
      wire#w1
      Contact( "HMI".Manu )
   END_RUNG wire#w2
   RUNG wire#w1
      Contact( "diBT_Reset" )
   END_RUNG wire#w2
   RUNG wire#powerrail
      Contact( "Variable".M_AutomaticModePermissionToCloseGrippers )
   END_RUNG wire#w3
   // the same network as SCL:
   "GripperOpenCloseAutoManu_DB1"(InAuto := "HMI".Auto,   // "GripperOpenCloseAutoManu"
                           InManu := "diPressOpenedUp" AND ("HMI".Manu OR "diBT_Reset"),
                           InGripperCloseManu := "HMI".CloseInManuGripper1,
                           InGripperOpenManu := "HMI".OpenInManuGripper1,
                           InGripperOpenAuto := "HMI".OpenInAutoGripper1,
                           InPressInjectionEnd := "diPressInjectionEnd",
                           InPinPresenceSE := "diSE_PresencePin1",
                           InGripperOpenedSE := "diSE_OpenGripper1",
                           InPermissinToClose := "Variable".M_AutomaticModePermissionToCloseGrippers,
                           EvGripperOutput => "Variable".M_EvGripperOutput1);
END_REGION

REGION Network 11: Electrovalve of Gripper 2
   // Sterowanie otwieraniem i zamykaniem chwytaka nr 2
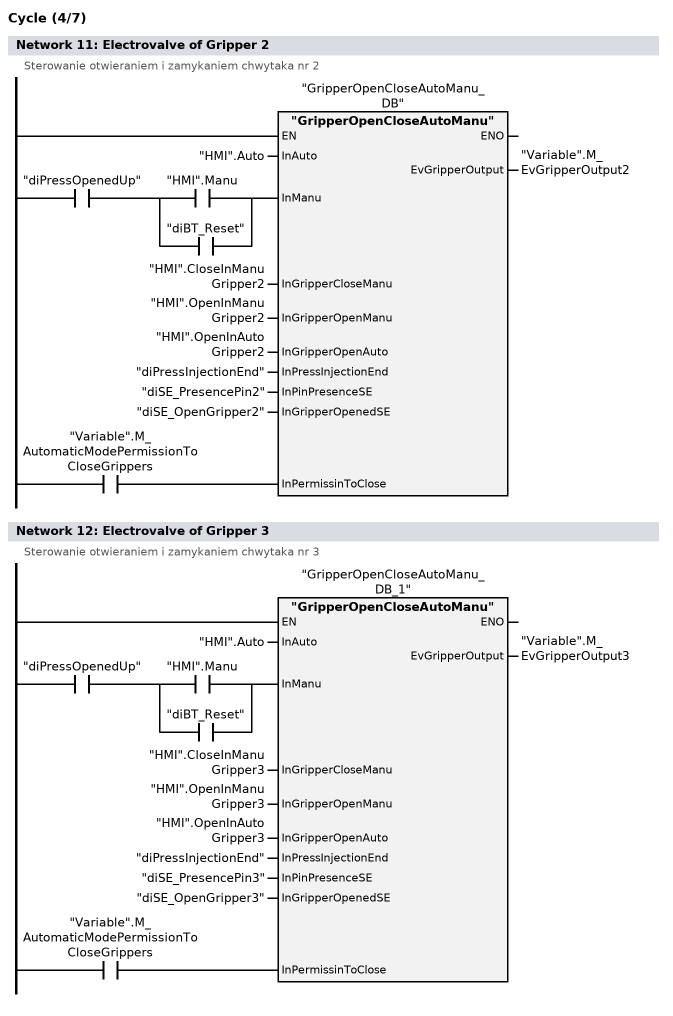
   RUNG wire#powerrail
      "GripperOpenCloseAutoManu_DB"(InManu := wire#w2, InPermissinToClose := wire#w3, InAuto := "HMI".Auto, InGripperCloseManu := "HMI".CloseInManuGripper2, InGripperOpenManu := "HMI".OpenInManuGripper2, InGripperOpenAuto := "HMI".OpenInAutoGripper2, InPressInjectionEnd := "diPressInjectionEnd", InPinPresenceSE := "diSE_PresencePin2", InGripperOpenedSE := "diSE_OpenGripper2", EvGripperOutput => "Variable".M_EvGripperOutput2)
   END_RUNG
   RUNG wire#powerrail
      Contact( "diPressOpenedUp" )
      wire#w1
      Contact( "HMI".Manu )
   END_RUNG wire#w2
   RUNG wire#w1
      Contact( "diBT_Reset" )
   END_RUNG wire#w2
   RUNG wire#powerrail
      Contact( "Variable".M_AutomaticModePermissionToCloseGrippers )
   END_RUNG wire#w3
   // the same network as SCL:
   "GripperOpenCloseAutoManu_DB"(InAuto := "HMI".Auto,   // "GripperOpenCloseAutoManu"
                           InManu := "diPressOpenedUp" AND ("HMI".Manu OR "diBT_Reset"),
                           InGripperCloseManu := "HMI".CloseInManuGripper2,
                           InGripperOpenManu := "HMI".OpenInManuGripper2,
                           InGripperOpenAuto := "HMI".OpenInAutoGripper2,
                           InPressInjectionEnd := "diPressInjectionEnd",
                           InPinPresenceSE := "diSE_PresencePin2",
                           InGripperOpenedSE := "diSE_OpenGripper2",
                           InPermissinToClose := "Variable".M_AutomaticModePermissionToCloseGrippers,
                           EvGripperOutput => "Variable".M_EvGripperOutput2);
END_REGION

REGION Network 12: Electrovalve of Gripper 3
   // Sterowanie otwieraniem i zamykaniem chwytaka nr 3
   RUNG wire#powerrail
      "GripperOpenCloseAutoManu_DB_1"(InManu := wire#w2, InPermissinToClose := wire#w3, InAuto := "HMI".Auto, InGripperCloseManu := "HMI".CloseInManuGripper3, InGripperOpenManu := "HMI".OpenInManuGripper3, InGripperOpenAuto := "HMI".OpenInAutoGripper3, InPressInjectionEnd := "diPressInjectionEnd", InPinPresenceSE := "diSE_PresencePin3", InGripperOpenedSE := "diSE_OpenGripper3", EvGripperOutput => "Variable".M_EvGripperOutput3)
   END_RUNG
   RUNG wire#powerrail
      Contact( "diPressOpenedUp" )
      wire#w1
      Contact( "HMI".Manu )
   END_RUNG wire#w2
   RUNG wire#w1
      Contact( "diBT_Reset" )
   END_RUNG wire#w2
   RUNG wire#powerrail
      Contact( "Variable".M_AutomaticModePermissionToCloseGrippers )
   END_RUNG wire#w3
   // the same network as SCL:
   "GripperOpenCloseAutoManu_DB_1"(InAuto := "HMI".Auto,   // "GripperOpenCloseAutoManu"
                           InManu := "diPressOpenedUp" AND ("HMI".Manu OR "diBT_Reset"),
                           InGripperCloseManu := "HMI".CloseInManuGripper3,
                           InGripperOpenManu := "HMI".OpenInManuGripper3,
                           InGripperOpenAuto := "HMI".OpenInAutoGripper3,
                           InPressInjectionEnd := "diPressInjectionEnd",
                           InPinPresenceSE := "diSE_PresencePin3",
                           InGripperOpenedSE := "diSE_OpenGripper3",
                           InPermissinToClose := "Variable".M_AutomaticModePermissionToCloseGrippers,
                           EvGripperOutput => "Variable".M_EvGripperOutput3);
END_REGION

REGION Network 13: Electrovalve of Gripper 4
   // Sterowanie otwieraniem i zamykaniem chwytaka nr 4
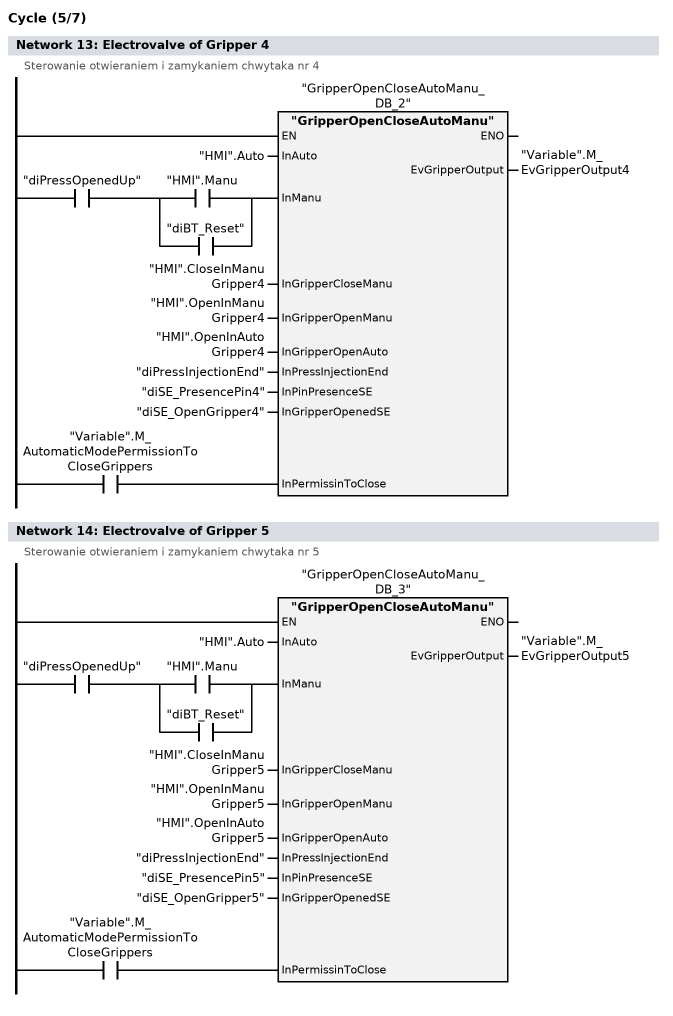
   RUNG wire#powerrail
      "GripperOpenCloseAutoManu_DB_2"(InManu := wire#w2, InPermissinToClose := wire#w3, InAuto := "HMI".Auto, InGripperCloseManu := "HMI".CloseInManuGripper4, InGripperOpenManu := "HMI".OpenInManuGripper4, InGripperOpenAuto := "HMI".OpenInAutoGripper4, InPressInjectionEnd := "diPressInjectionEnd", InPinPresenceSE := "diSE_PresencePin4", InGripperOpenedSE := "diSE_OpenGripper4", EvGripperOutput => "Variable".M_EvGripperOutput4)
   END_RUNG
   RUNG wire#powerrail
      Contact( "diPressOpenedUp" )
      wire#w1
      Contact( "HMI".Manu )
   END_RUNG wire#w2
   RUNG wire#w1
      Contact( "diBT_Reset" )
   END_RUNG wire#w2
   RUNG wire#powerrail
      Contact( "Variable".M_AutomaticModePermissionToCloseGrippers )
   END_RUNG wire#w3
   // the same network as SCL:
   "GripperOpenCloseAutoManu_DB_2"(InAuto := "HMI".Auto,   // "GripperOpenCloseAutoManu"
                           InManu := "diPressOpenedUp" AND ("HMI".Manu OR "diBT_Reset"),
                           InGripperCloseManu := "HMI".CloseInManuGripper4,
                           InGripperOpenManu := "HMI".OpenInManuGripper4,
                           InGripperOpenAuto := "HMI".OpenInAutoGripper4,
                           InPressInjectionEnd := "diPressInjectionEnd",
                           InPinPresenceSE := "diSE_PresencePin4",
                           InGripperOpenedSE := "diSE_OpenGripper4",
                           InPermissinToClose := "Variable".M_AutomaticModePermissionToCloseGrippers,
                           EvGripperOutput => "Variable".M_EvGripperOutput4);
END_REGION

REGION Network 14: Electrovalve of Gripper 5
   // Sterowanie otwieraniem i zamykaniem chwytaka nr 5
   RUNG wire#powerrail
      "GripperOpenCloseAutoManu_DB_3"(InManu := wire#w2, InPermissinToClose := wire#w3, InAuto := "HMI".Auto, InGripperCloseManu := "HMI".CloseInManuGripper5, InGripperOpenManu := "HMI".OpenInManuGripper5, InGripperOpenAuto := "HMI".OpenInAutoGripper5, InPressInjectionEnd := "diPressInjectionEnd", InPinPresenceSE := "diSE_PresencePin5", InGripperOpenedSE := "diSE_OpenGripper5", EvGripperOutput => "Variable".M_EvGripperOutput5)
   END_RUNG
   RUNG wire#powerrail
      Contact( "diPressOpenedUp" )
      wire#w1
      Contact( "HMI".Manu )
   END_RUNG wire#w2
   RUNG wire#w1
      Contact( "diBT_Reset" )
   END_RUNG wire#w2
   RUNG wire#powerrail
      Contact( "Variable".M_AutomaticModePermissionToCloseGrippers )
   END_RUNG wire#w3
   // the same network as SCL:
   "GripperOpenCloseAutoManu_DB_3"(InAuto := "HMI".Auto,   // "GripperOpenCloseAutoManu"
                           InManu := "diPressOpenedUp" AND ("HMI".Manu OR "diBT_Reset"),
                           InGripperCloseManu := "HMI".CloseInManuGripper5,
                           InGripperOpenManu := "HMI".OpenInManuGripper5,
                           InGripperOpenAuto := "HMI".OpenInAutoGripper5,
                           InPressInjectionEnd := "diPressInjectionEnd",
                           InPinPresenceSE := "diSE_PresencePin5",
                           InGripperOpenedSE := "diSE_OpenGripper5",
                           InPermissinToClose := "Variable".M_AutomaticModePermissionToCloseGrippers,
                           EvGripperOutput => "Variable".M_EvGripperOutput5);
END_REGION

REGION Network 15: Electrovalve of Gripper 6
   // Sterowanie otwieraniem i zamykaniem chwytaka nr 6
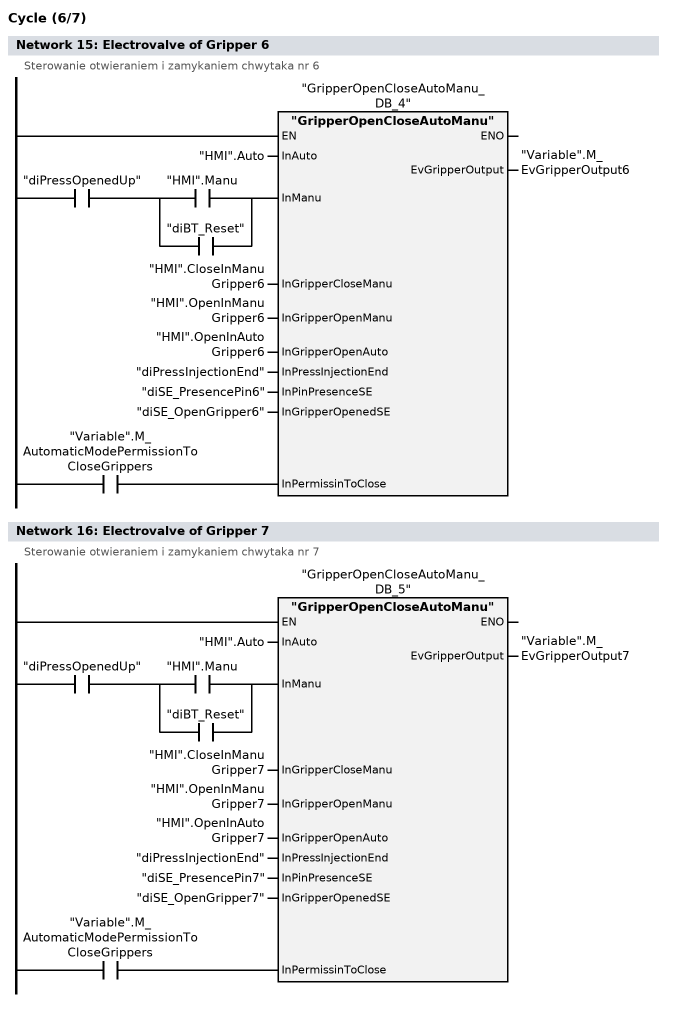
   RUNG wire#powerrail
      "GripperOpenCloseAutoManu_DB_4"(InManu := wire#w2, InPermissinToClose := wire#w3, InAuto := "HMI".Auto, InGripperCloseManu := "HMI".CloseInManuGripper6, InGripperOpenManu := "HMI".OpenInManuGripper6, InGripperOpenAuto := "HMI".OpenInAutoGripper6, InPressInjectionEnd := "diPressInjectionEnd", InPinPresenceSE := "diSE_PresencePin6", InGripperOpenedSE := "diSE_OpenGripper6", EvGripperOutput => "Variable".M_EvGripperOutput6)
   END_RUNG
   RUNG wire#powerrail
      Contact( "diPressOpenedUp" )
      wire#w1
      Contact( "HMI".Manu )
   END_RUNG wire#w2
   RUNG wire#w1
      Contact( "diBT_Reset" )
   END_RUNG wire#w2
   RUNG wire#powerrail
      Contact( "Variable".M_AutomaticModePermissionToCloseGrippers )
   END_RUNG wire#w3
   // the same network as SCL:
   "GripperOpenCloseAutoManu_DB_4"(InAuto := "HMI".Auto,   // "GripperOpenCloseAutoManu"
                           InManu := "diPressOpenedUp" AND ("HMI".Manu OR "diBT_Reset"),
                           InGripperCloseManu := "HMI".CloseInManuGripper6,
                           InGripperOpenManu := "HMI".OpenInManuGripper6,
                           InGripperOpenAuto := "HMI".OpenInAutoGripper6,
                           InPressInjectionEnd := "diPressInjectionEnd",
                           InPinPresenceSE := "diSE_PresencePin6",
                           InGripperOpenedSE := "diSE_OpenGripper6",
                           InPermissinToClose := "Variable".M_AutomaticModePermissionToCloseGrippers,
                           EvGripperOutput => "Variable".M_EvGripperOutput6);
END_REGION

REGION Network 16: Electrovalve of Gripper 7
   // Sterowanie otwieraniem i zamykaniem chwytaka nr 7
   RUNG wire#powerrail
      "GripperOpenCloseAutoManu_DB_5"(InManu := wire#w2, InPermissinToClose := wire#w3, InAuto := "HMI".Auto, InGripperCloseManu := "HMI".CloseInManuGripper7, InGripperOpenManu := "HMI".OpenInManuGripper7, InGripperOpenAuto := "HMI".OpenInAutoGripper7, InPressInjectionEnd := "diPressInjectionEnd", InPinPresenceSE := "diSE_PresencePin7", InGripperOpenedSE := "diSE_OpenGripper7", EvGripperOutput => "Variable".M_EvGripperOutput7)
   END_RUNG
   RUNG wire#powerrail
      Contact( "diPressOpenedUp" )
      wire#w1
      Contact( "HMI".Manu )
   END_RUNG wire#w2
   RUNG wire#w1
      Contact( "diBT_Reset" )
   END_RUNG wire#w2
   RUNG wire#powerrail
      Contact( "Variable".M_AutomaticModePermissionToCloseGrippers )
   END_RUNG wire#w3
   // the same network as SCL:
   "GripperOpenCloseAutoManu_DB_5"(InAuto := "HMI".Auto,   // "GripperOpenCloseAutoManu"
                           InManu := "diPressOpenedUp" AND ("HMI".Manu OR "diBT_Reset"),
                           InGripperCloseManu := "HMI".CloseInManuGripper7,
                           InGripperOpenManu := "HMI".OpenInManuGripper7,
                           InGripperOpenAuto := "HMI".OpenInAutoGripper7,
                           InPressInjectionEnd := "diPressInjectionEnd",
                           InPinPresenceSE := "diSE_PresencePin7",
                           InGripperOpenedSE := "diSE_OpenGripper7",
                           InPermissinToClose := "Variable".M_AutomaticModePermissionToCloseGrippers,
                           EvGripperOutput => "Variable".M_EvGripperOutput7);
END_REGION

REGION Network 17: Electrovalve of Gripper 8
   // Sterowanie otwieraniem i zamykaniem chwytaka nr 8
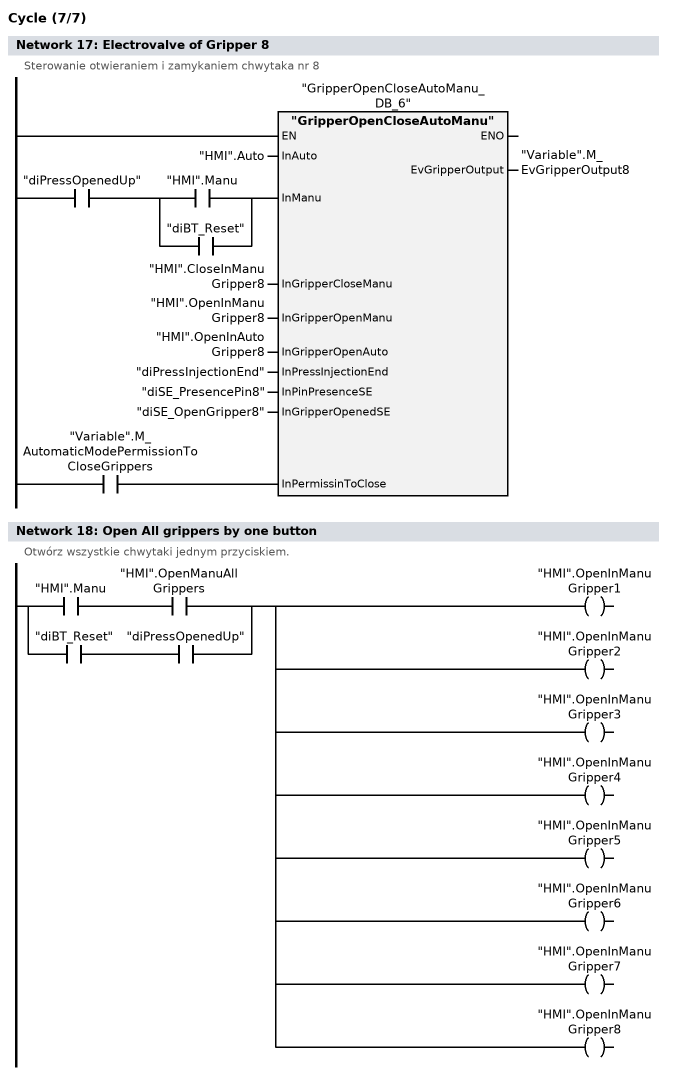
   RUNG wire#powerrail
      "GripperOpenCloseAutoManu_DB_6"(InManu := wire#w2, InPermissinToClose := wire#w3, InAuto := "HMI".Auto, InGripperCloseManu := "HMI".CloseInManuGripper8, InGripperOpenManu := "HMI".OpenInManuGripper8, InGripperOpenAuto := "HMI".OpenInAutoGripper8, InPressInjectionEnd := "diPressInjectionEnd", InPinPresenceSE := "diSE_PresencePin8", InGripperOpenedSE := "diSE_OpenGripper8", EvGripperOutput => "Variable".M_EvGripperOutput8)
   END_RUNG
   RUNG wire#powerrail
      Contact( "diPressOpenedUp" )
      wire#w1
      Contact( "HMI".Manu )
   END_RUNG wire#w2
   RUNG wire#w1
      Contact( "diBT_Reset" )
   END_RUNG wire#w2
   RUNG wire#powerrail
      Contact( "Variable".M_AutomaticModePermissionToCloseGrippers )
   END_RUNG wire#w3
   // the same network as SCL:
   "GripperOpenCloseAutoManu_DB_6"(InAuto := "HMI".Auto,   // "GripperOpenCloseAutoManu"
                           InManu := "diPressOpenedUp" AND ("HMI".Manu OR "diBT_Reset"),
                           InGripperCloseManu := "HMI".CloseInManuGripper8,
                           InGripperOpenManu := "HMI".OpenInManuGripper8,
                           InGripperOpenAuto := "HMI".OpenInAutoGripper8,
                           InPressInjectionEnd := "diPressInjectionEnd",
                           InPinPresenceSE := "diSE_PresencePin8",
                           InGripperOpenedSE := "diSE_OpenGripper8",
                           InPermissinToClose := "Variable".M_AutomaticModePermissionToCloseGrippers,
                           EvGripperOutput => "Variable".M_EvGripperOutput8);
END_REGION

REGION Network 18: Open All grippers by one button
   // Otwórz wszystkie chwytaki jednym przyciskiem.
   RUNG wire#powerrail
      Contact( "HMI".Manu )
      Contact( "HMI".OpenManuAllGrippers )
      wire#w1
      Coil( "HMI".OpenInManuGripper1 )
   END_RUNG
   RUNG wire#powerrail
      Contact( "diBT_Reset" )
      Contact( "diPressOpenedUp" )
   END_RUNG wire#w1
   RUNG wire#w1
      Coil( "HMI".OpenInManuGripper2 )
   END_RUNG
   RUNG wire#w1
      Coil( "HMI".OpenInManuGripper3 )
   END_RUNG
   RUNG wire#w1
      Coil( "HMI".OpenInManuGripper4 )
   END_RUNG
   RUNG wire#w1
      Coil( "HMI".OpenInManuGripper5 )
   END_RUNG
   RUNG wire#w1
      Coil( "HMI".OpenInManuGripper6 )
   END_RUNG
   RUNG wire#w1
      Coil( "HMI".OpenInManuGripper7 )
   END_RUNG
   RUNG wire#w1
      Coil( "HMI".OpenInManuGripper8 )
   END_RUNG
   // the same network as SCL:
   "HMI".OpenInManuGripper1 := ("HMI".Manu AND "HMI".OpenManuAllGrippers) OR ("diBT_Reset" AND "diPressOpenedUp");
   "HMI".OpenInManuGripper2 := "HMI".OpenInManuGripper1;
   "HMI".OpenInManuGripper3 := "HMI".OpenInManuGripper1;
   "HMI".OpenInManuGripper4 := "HMI".OpenInManuGripper1;
   "HMI".OpenInManuGripper5 := "HMI".OpenInManuGripper1;
   "HMI".OpenInManuGripper6 := "HMI".OpenInManuGripper1;
   "HMI".OpenInManuGripper7 := "HMI".OpenInManuGripper1;
   "HMI".OpenInManuGripper8 := "HMI".OpenInManuGripper1;
END_REGION
END_FUNCTION

FUNCTION "Alarms" : Void   // FC2, LAD
{ S7_Optimized_Access := 'TRUE' }
VERSION : 0.1
   VAR CONSTANT
      DELAY_TO_GRIPPER_ALARM : Time := T#5s;
   END_VAR
BEGIN

REGION Network 1: An alarm of left actuator of table - grippers
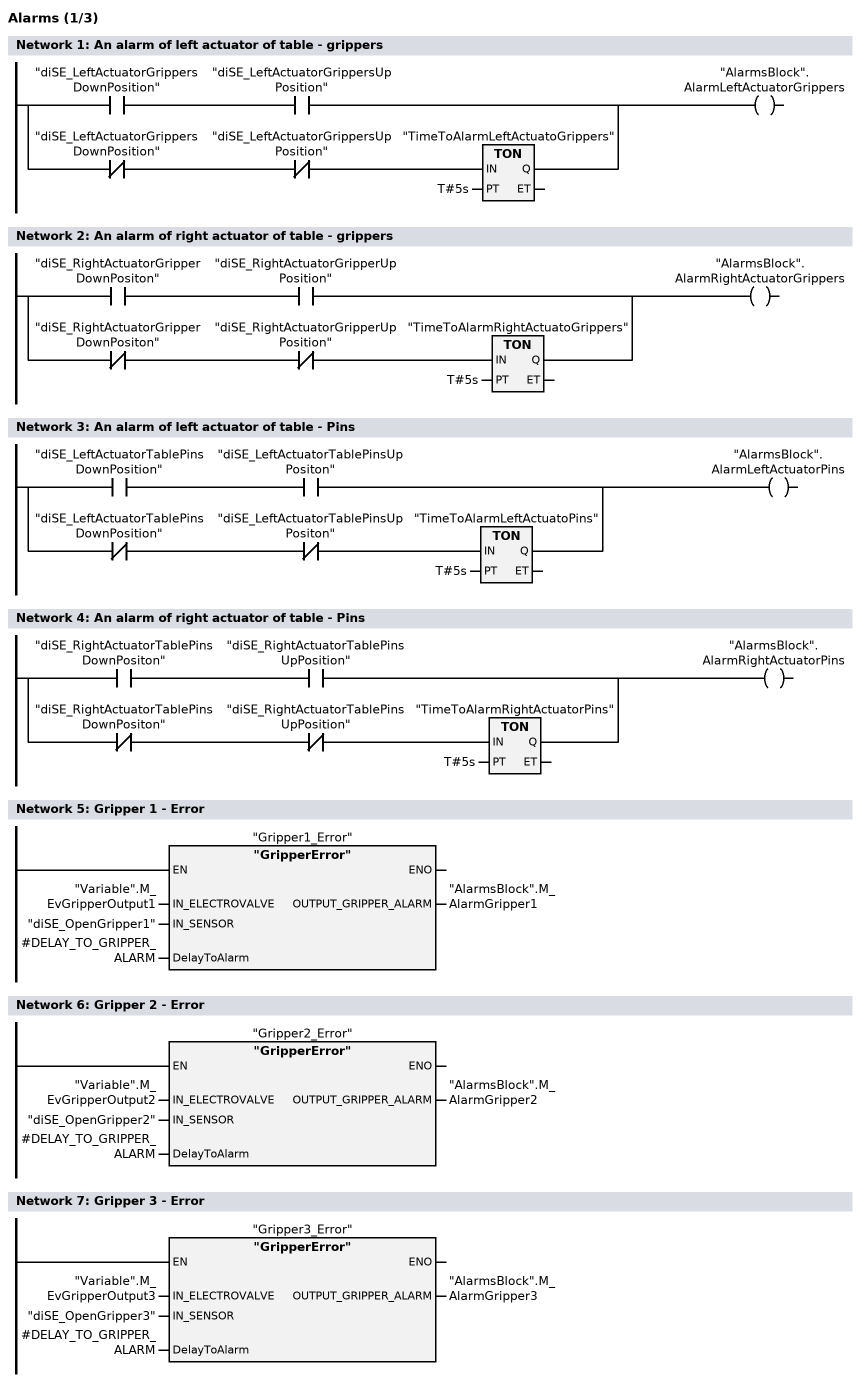
   "TimeToAlarmLeftActuatoGrippers".TON(IN := NOT "diSE_LeftActuatorGrippersDownPosition" AND NOT "diSE_LeftActuatorGrippersUpPosition",
                           PT := T#5s);
   "AlarmsBlock".AlarmLeftActuatorGrippers := ("diSE_LeftActuatorGrippersDownPosition" AND "diSE_LeftActuatorGrippersUpPosition") OR "TimeToAlarmLeftActuatoGrippers".Q;
END_REGION

REGION Network 2: An alarm of right actuator of table - grippers
   "TimeToAlarmRightActuatoGrippers".TON(IN := NOT "diSE_RightActuatorGripperDownPositon" AND NOT "diSE_RightActuatorGripperUpPosition",
                           PT := T#5s);
   "AlarmsBlock".AlarmRightActuatorGrippers := ("diSE_RightActuatorGripperDownPositon" AND "diSE_RightActuatorGripperUpPosition") OR "TimeToAlarmRightActuatoGrippers".Q;
END_REGION

REGION Network 3: An alarm of left actuator of table - Pins
   "TimeToAlarmLeftActuatoPins".TON(IN := NOT "diSE_LeftActuatorTablePinsDownPosition" AND NOT "diSE_LeftActuatorTablePinsUpPositon",
                           PT := T#5s);
   "AlarmsBlock".AlarmLeftActuatorPins := ("diSE_LeftActuatorTablePinsDownPosition" AND "diSE_LeftActuatorTablePinsUpPositon") OR "TimeToAlarmLeftActuatoPins".Q;
END_REGION

REGION Network 4: An alarm of right actuator of table - Pins
   "TimeToAlarmRightActuatorPins".TON(IN := NOT "diSE_RightActuatorTablePinsDownPositon" AND NOT "diSE_RightActuatorTablePinsUpPosition",
                           PT := T#5s);
   "AlarmsBlock".AlarmRightActuatorPins := ("diSE_RightActuatorTablePinsDownPositon" AND "diSE_RightActuatorTablePinsUpPosition") OR "TimeToAlarmRightActuatorPins".Q;
END_REGION

REGION Network 5: Gripper 1 - Error
   RUNG wire#powerrail
      "Gripper1_Error"(IN_ELECTROVALVE := "Variable".M_EvGripperOutput1, IN_SENSOR := "diSE_OpenGripper1", DelayToAlarm := #DELAY_TO_GRIPPER_ALARM, OUTPUT_GRIPPER_ALARM => "AlarmsBlock".M_AlarmGripper1)
   END_RUNG
   // the same network as SCL:
   "Gripper1_Error"(IN_ELECTROVALVE := "Variable".M_EvGripperOutput1,   // "GripperError"
                    IN_SENSOR := "diSE_OpenGripper1",
                    DelayToAlarm := #DELAY_TO_GRIPPER_ALARM,
                    OUTPUT_GRIPPER_ALARM => "AlarmsBlock".M_AlarmGripper1);
END_REGION

REGION Network 6: Gripper 2 - Error
   RUNG wire#powerrail
      "Gripper2_Error"(IN_ELECTROVALVE := "Variable".M_EvGripperOutput2, IN_SENSOR := "diSE_OpenGripper2", DelayToAlarm := #DELAY_TO_GRIPPER_ALARM, OUTPUT_GRIPPER_ALARM => "AlarmsBlock".M_AlarmGripper2)
   END_RUNG
   // the same network as SCL:
   "Gripper2_Error"(IN_ELECTROVALVE := "Variable".M_EvGripperOutput2,   // "GripperError"
                    IN_SENSOR := "diSE_OpenGripper2",
                    DelayToAlarm := #DELAY_TO_GRIPPER_ALARM,
                    OUTPUT_GRIPPER_ALARM => "AlarmsBlock".M_AlarmGripper2);
END_REGION

REGION Network 7: Gripper 3 - Error
   RUNG wire#powerrail
      "Gripper3_Error"(IN_ELECTROVALVE := "Variable".M_EvGripperOutput3, IN_SENSOR := "diSE_OpenGripper3", DelayToAlarm := #DELAY_TO_GRIPPER_ALARM, OUTPUT_GRIPPER_ALARM => "AlarmsBlock".M_AlarmGripper3)
   END_RUNG
   // the same network as SCL:
   "Gripper3_Error"(IN_ELECTROVALVE := "Variable".M_EvGripperOutput3,   // "GripperError"
                    IN_SENSOR := "diSE_OpenGripper3",
                    DelayToAlarm := #DELAY_TO_GRIPPER_ALARM,
                    OUTPUT_GRIPPER_ALARM => "AlarmsBlock".M_AlarmGripper3);
END_REGION

REGION Network 8: Gripper 4 - Error
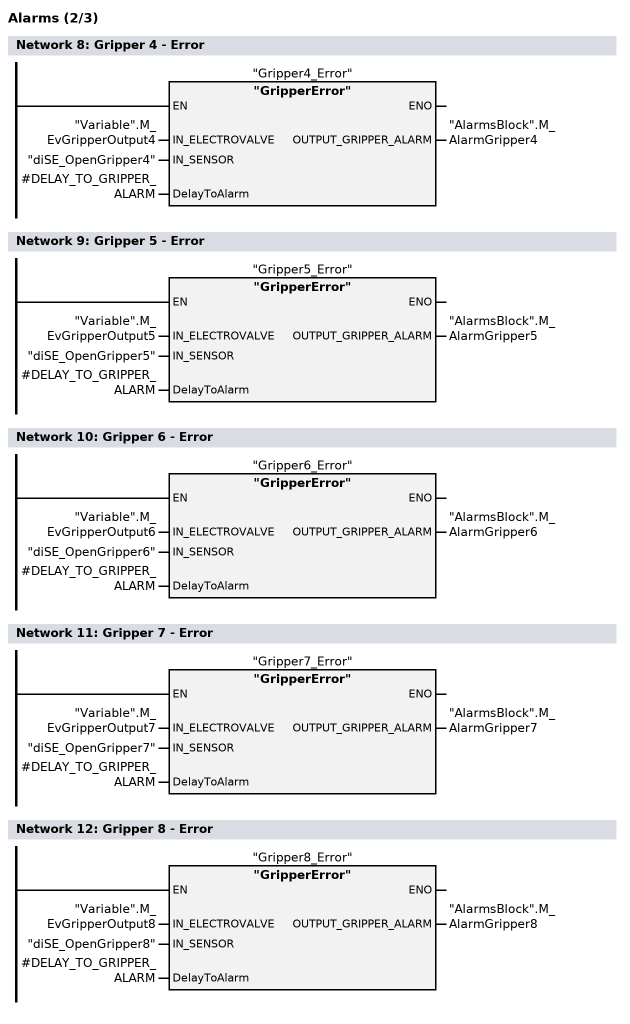
   RUNG wire#powerrail
      "Gripper4_Error"(IN_ELECTROVALVE := "Variable".M_EvGripperOutput4, IN_SENSOR := "diSE_OpenGripper4", DelayToAlarm := #DELAY_TO_GRIPPER_ALARM, OUTPUT_GRIPPER_ALARM => "AlarmsBlock".M_AlarmGripper4)
   END_RUNG
   // the same network as SCL:
   "Gripper4_Error"(IN_ELECTROVALVE := "Variable".M_EvGripperOutput4,   // "GripperError"
                    IN_SENSOR := "diSE_OpenGripper4",
                    DelayToAlarm := #DELAY_TO_GRIPPER_ALARM,
                    OUTPUT_GRIPPER_ALARM => "AlarmsBlock".M_AlarmGripper4);
END_REGION

REGION Network 9: Gripper 5 - Error
   RUNG wire#powerrail
      "Gripper5_Error"(IN_ELECTROVALVE := "Variable".M_EvGripperOutput5, IN_SENSOR := "diSE_OpenGripper5", DelayToAlarm := #DELAY_TO_GRIPPER_ALARM, OUTPUT_GRIPPER_ALARM => "AlarmsBlock".M_AlarmGripper5)
   END_RUNG
   // the same network as SCL:
   "Gripper5_Error"(IN_ELECTROVALVE := "Variable".M_EvGripperOutput5,   // "GripperError"
                    IN_SENSOR := "diSE_OpenGripper5",
                    DelayToAlarm := #DELAY_TO_GRIPPER_ALARM,
                    OUTPUT_GRIPPER_ALARM => "AlarmsBlock".M_AlarmGripper5);
END_REGION

REGION Network 10: Gripper 6 - Error
   RUNG wire#powerrail
      "Gripper6_Error"(IN_ELECTROVALVE := "Variable".M_EvGripperOutput6, IN_SENSOR := "diSE_OpenGripper6", DelayToAlarm := #DELAY_TO_GRIPPER_ALARM, OUTPUT_GRIPPER_ALARM => "AlarmsBlock".M_AlarmGripper6)
   END_RUNG
   // the same network as SCL:
   "Gripper6_Error"(IN_ELECTROVALVE := "Variable".M_EvGripperOutput6,   // "GripperError"
                    IN_SENSOR := "diSE_OpenGripper6",
                    DelayToAlarm := #DELAY_TO_GRIPPER_ALARM,
                    OUTPUT_GRIPPER_ALARM => "AlarmsBlock".M_AlarmGripper6);
END_REGION

REGION Network 11: Gripper 7 - Error
   RUNG wire#powerrail
      "Gripper7_Error"(IN_ELECTROVALVE := "Variable".M_EvGripperOutput7, IN_SENSOR := "diSE_OpenGripper7", DelayToAlarm := #DELAY_TO_GRIPPER_ALARM, OUTPUT_GRIPPER_ALARM => "AlarmsBlock".M_AlarmGripper7)
   END_RUNG
   // the same network as SCL:
   "Gripper7_Error"(IN_ELECTROVALVE := "Variable".M_EvGripperOutput7,   // "GripperError"
                    IN_SENSOR := "diSE_OpenGripper7",
                    DelayToAlarm := #DELAY_TO_GRIPPER_ALARM,
                    OUTPUT_GRIPPER_ALARM => "AlarmsBlock".M_AlarmGripper7);
END_REGION

REGION Network 12: Gripper 8 - Error
   RUNG wire#powerrail
      "Gripper8_Error"(IN_ELECTROVALVE := "Variable".M_EvGripperOutput8, IN_SENSOR := "diSE_OpenGripper8", DelayToAlarm := #DELAY_TO_GRIPPER_ALARM, OUTPUT_GRIPPER_ALARM => "AlarmsBlock".M_AlarmGripper8)
   END_RUNG
   // the same network as SCL:
   "Gripper8_Error"(IN_ELECTROVALVE := "Variable".M_EvGripperOutput8,   // "GripperError"
                    IN_SENSOR := "diSE_OpenGripper8",
                    DelayToAlarm := #DELAY_TO_GRIPPER_ALARM,
                    OUTPUT_GRIPPER_ALARM => "AlarmsBlock".M_AlarmGripper8);
END_REGION

REGION Network 13: An alarm occur
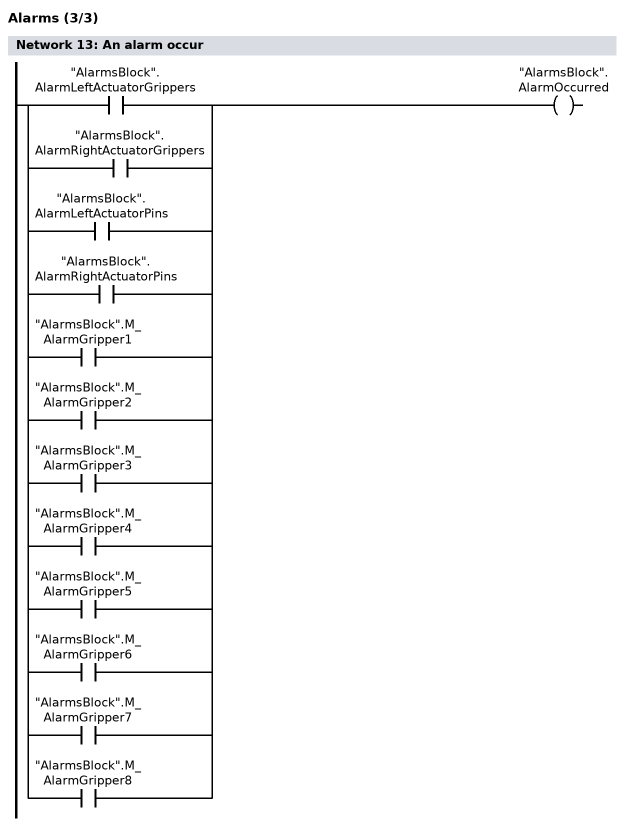
   RUNG wire#powerrail
      Contact( "AlarmsBlock".AlarmLeftActuatorGrippers )
      wire#w1
      Coil( "AlarmsBlock".AlarmOccurred )
   END_RUNG
   RUNG wire#powerrail
      Contact( "AlarmsBlock".AlarmRightActuatorGrippers )
   END_RUNG wire#w1
   RUNG wire#powerrail
      Contact( "AlarmsBlock".AlarmLeftActuatorPins )
   END_RUNG wire#w1
   RUNG wire#powerrail
      Contact( "AlarmsBlock".AlarmRightActuatorPins )
   END_RUNG wire#w1
   RUNG wire#powerrail
      Contact( "AlarmsBlock".M_AlarmGripper1 )
   END_RUNG wire#w1
   RUNG wire#powerrail
      Contact( "AlarmsBlock".M_AlarmGripper2 )
   END_RUNG wire#w1
   RUNG wire#powerrail
      Contact( "AlarmsBlock".M_AlarmGripper3 )
   END_RUNG wire#w1
   RUNG wire#powerrail
      Contact( "AlarmsBlock".M_AlarmGripper4 )
   END_RUNG wire#w1
   RUNG wire#powerrail
      Contact( "AlarmsBlock".M_AlarmGripper5 )
   END_RUNG wire#w1
   RUNG wire#powerrail
      Contact( "AlarmsBlock".M_AlarmGripper6 )
   END_RUNG wire#w1
   RUNG wire#powerrail
      Contact( "AlarmsBlock".M_AlarmGripper7 )
   END_RUNG wire#w1
   RUNG wire#powerrail
      Contact( "AlarmsBlock".M_AlarmGripper8 )
   END_RUNG wire#w1
   // the same network as SCL:
   "AlarmsBlock".AlarmOccurred := "AlarmsBlock".AlarmLeftActuatorGrippers OR "AlarmsBlock".AlarmRightActuatorGrippers OR "AlarmsBlock".AlarmLeftActuatorPins OR "AlarmsBlock".AlarmRightActuatorPins OR "AlarmsBlock".M_AlarmGripper1 OR "AlarmsBlock".M_AlarmGripper2 OR "AlarmsBlock".M_AlarmGripper3 OR "AlarmsBlock".M_AlarmGripper4 OR "AlarmsBlock".M_AlarmGripper5 OR "AlarmsBlock".M_AlarmGripper6 OR "AlarmsBlock".M_AlarmGripper7 OR "AlarmsBlock".M_AlarmGripper8;
END_REGION
END_FUNCTION

ORGANIZATION_BLOCK "Main"   // OB1, SCL, ProgramCycle
TITLE = "Main Program Sweep (Cycle)"
{ S7_Optimized_Access := 'TRUE' }
VERSION : 0.1
   VAR_INPUT
      Initial_Call : Bool;   // Initial call of this OB
      Remanence : Bool;   // =True, if remanent data are available
   END_VAR
BEGIN
   "Cycle"();
   "Alarms"();
   "Outputs_DB"();
END_ORGANIZATION_BLOCK

// folder: MyFunctions

FUNCTION_BLOCK "ElectricValve"   // FB1, SCL
{ S7_Optimized_Access := 'TRUE' }
VERSION : 0.1
   VAR_INPUT
      InputControlValve : Bool;
   END_VAR
   VAR_OUTPUT
      ValveUp_Open : Bool;
      ValveDown_Close : Bool;
   END_VAR
BEGIN

   IF #InputControlValve THEN
       #ValveUp_Open := FALSE;
       #ValveDown_Close := TRUE;
   ELSE
       #ValveUp_Open := TRUE;
       #ValveDown_Close := FALSE;
   END_IF;
END_FUNCTION_BLOCK

FUNCTION_BLOCK "Buzzer"   // FB3, SCL
{ S7_Optimized_Access := 'TRUE' }
VERSION : 0.1
   VAR_INPUT
      INPUT : Bool;
      TimeOfSignal : Time;
   END_VAR
   VAR_OUTPUT
      BuzzerActivationOutput : Bool;
   END_VAR
   VAR RETAIN
      TimeOfBuzzerSignal : TP_TIME;
   END_VAR
BEGIN

   //Buzzer activation for programing time.

       #TimeOfBuzzerSignal(IN := #INPUT,
                           PT := #TimeOfSignal);
       #BuzzerActivationOutput := #TimeOfBuzzerSignal.Q;
END_FUNCTION_BLOCK

FUNCTION_BLOCK "GripperError"   // FB4, SCL
{ S7_Optimized_Access := 'TRUE' }
VERSION : 0.1
   VAR_INPUT
      IN_ELECTROVALVE : Bool;
      IN_SENSOR : Bool;
      DelayToAlarm : Time;
   END_VAR
   VAR_OUTPUT
      OUTPUT_GRIPPER_ALARM : Bool;
   END_VAR
   VAR
      MarkerOutputGripperAlarm : Bool;
      IEC_Timer_0_Instance : TON_TIME;
   END_VAR
BEGIN

   //If command electrovalve of gripper is ON and sensor of gripper is still ON, then alarm occurring.
   //Jeśli wystawiony jest sygnał załączenia elektrozaworu chwytaki i czujnik chwytaka jest wciąż aktywny
   //to załączany jest alarm chwytaka.
   //
   IF #IN_ELECTROVALVE AND #IN_SENSOR THEN
       // Statement section IF
       #MarkerOutputGripperAlarm := TRUE;
   ELSIF
       (NOT #IN_ELECTROVALVE)AND (NOT #IN_SENSOR)THEN
       #MarkerOutputGripperAlarm := TRUE;

   ELSE
       #MarkerOutputGripperAlarm := FALSE;
   END_IF;

   #IEC_Timer_0_Instance(IN:=#MarkerOutputGripperAlarm,PT:=#DelayToAlarm);
   #OUTPUT_GRIPPER_ALARM := #IEC_Timer_0_Instance.Q;
END_FUNCTION_BLOCK

FUNCTION_BLOCK "GripperOpenCloseAutoManu"   // FB5, LAD
{ S7_Optimized_Access := 'TRUE' }
   VAR_INPUT
      InAuto : Bool;
      InManu : Bool;
      InGripperCloseManu : Bool;
      InGripperOpenManu : Bool;
      InGripperOpenAuto : Bool;
      InPressInjectionEnd : Bool;
      InPinPresenceSE : Bool;
      InGripperOpenedSE : Bool;
      InPermissinToClose : Bool;
   END_VAR
   VAR_OUTPUT
      EvGripperOutput : Bool;
   END_VAR
BEGIN

REGION Network 2: Electrovalve of Gripper
   // Sterowanie otwieraniem i zamykaniem chwytaka
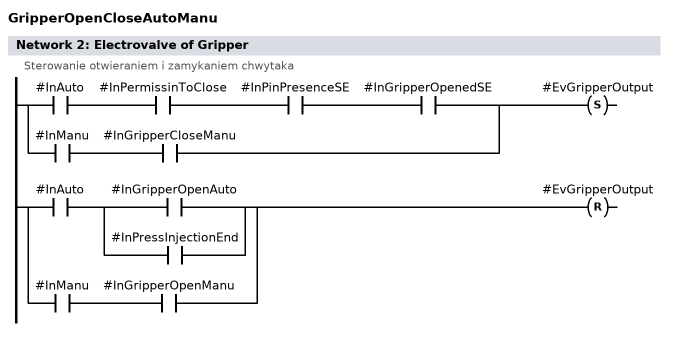
   RUNG wire#powerrail
      Contact( #InAuto )
      Contact( #InPermissinToClose )
      Contact( #InPinPresenceSE )
      Contact( #InGripperOpenedSE )
      wire#w1
      S_Coil( #EvGripperOutput )
   END_RUNG
   RUNG wire#powerrail
      Contact( #InManu )
      Contact( #InGripperCloseManu )
   END_RUNG wire#w1
   RUNG wire#powerrail
      Contact( #InAuto )
      wire#w2
      Contact( #InGripperOpenAuto )
      wire#w3
      R_Coil( #EvGripperOutput )
   END_RUNG
   RUNG wire#w2
      Contact( #InPressInjectionEnd )
   END_RUNG wire#w3
   RUNG wire#powerrail
      Contact( #InManu )
      Contact( #InGripperOpenManu )
   END_RUNG wire#w3
   // the same network as SCL:
   IF (#InAuto AND #InPermissinToClose AND #InPinPresenceSE AND #InGripperOpenedSE) OR (#InManu AND #InGripperCloseManu) THEN
       #EvGripperOutput := TRUE;
   END_IF;
   IF (#InAuto AND (#InGripperOpenAuto OR #InPressInjectionEnd)) OR (#InManu AND #InGripperOpenManu) THEN
       #EvGripperOutput := FALSE;
   END_IF;
END_REGION
END_FUNCTION_BLOCK

(* ===== HMI "HMI_RT_1" =====
system functions are stored by id; their names below are inferred from use
connection "HMI_Connection_1": ETHERNET, SMART_S7_1200_OMS

HMI tags "HMI"
   "HMI_Auto" : Bool = PLC HMI.Auto AT %DB8.DBX0.0, 100 ms
   "HMI_Manu" : Bool = PLC HMI.Manu AT %DB8.DBX0.1, 100 ms
   "HMI_OpenInAutoGripper1" : Bool = PLC HMI.OpenInAutoGripper1 AT %DB8.DBX0.2, 100 ms
   "HMI_OpenInAutoGripper2" : Bool = PLC HMI.OpenInAutoGripper2 AT %DB8.DBX0.3, 100 ms
   "HMI_OpenInAutoGripper3" : Bool = PLC HMI.OpenInAutoGripper3 AT %DB8.DBX0.4, 100 ms
   "HMI_OpenInAutoGripper4" : Bool = PLC HMI.OpenInAutoGripper4 AT %DB8.DBX0.5, 100 ms
   "HMI_OpenInAutoGripper5" : Bool = PLC HMI.OpenInAutoGripper5 AT %DB8.DBX0.6, 100 ms
   "HMI_OpenInAutoGripper6" : Bool = PLC HMI.OpenInAutoGripper6 AT %DB8.DBX0.7, 100 ms
   "HMI_OpenInAutoGripper7" : Bool = PLC HMI.OpenInAutoGripper7 AT %DB8.DBX1.0, 100 ms
   "HMI_OpenInAutoGripper8" : Bool = PLC HMI.OpenInAutoGripper8 AT %DB8.DBX1.1, 100 ms
   "HMI_OpenInManuGripper1" : Bool = PLC HMI.OpenInManuGripper1 AT %DB8.DBX1.2, 100 ms
   "HMI_OpenInManuGripper2" : Bool = PLC HMI.OpenInManuGripper2 AT %DB8.DBX1.3, 100 ms
   "HMI_OpenInManuGripper3" : Bool = PLC HMI.OpenInManuGripper3 AT %DB8.DBX1.4, 100 ms
   "HMI_OpenInManuGripper4" : Bool = PLC HMI.OpenInManuGripper4 AT %DB8.DBX1.5, 100 ms
   "HMI_OpenInManuGripper5" : Bool = PLC HMI.OpenInManuGripper5 AT %DB8.DBX1.6, 100 ms
   "HMI_OpenInManuGripper6" : Bool = PLC HMI.OpenInManuGripper6 AT %DB8.DBX1.7, 100 ms
   "HMI_OpenInManuGripper7" : Bool = PLC HMI.OpenInManuGripper7 AT %DB8.DBX2.0, 100 ms
   "HMI_OpenInManuGripper8" : Bool = PLC HMI.OpenInManuGripper8 AT %DB8.DBX2.1, 100 ms
   "HMI_CloseInManuGripper1" : Bool = PLC HMI.CloseInManuGripper1 AT %DB8.DBX2.2, 100 ms
   "HMI_CloseInManuGripper2" : Bool = PLC HMI.CloseInManuGripper2 AT %DB8.DBX2.3, 100 ms
   "HMI_CloseInManuGripper3" : Bool = PLC HMI.CloseInManuGripper3 AT %DB8.DBX2.4, 100 ms
   "HMI_CloseInManuGripper4" : Bool = PLC HMI.CloseInManuGripper4 AT %DB8.DBX2.5, 100 ms
   "HMI_CloseInManuGripper5" : Bool = PLC HMI.CloseInManuGripper5 AT %DB8.DBX2.6, 100 ms
   "HMI_CloseInManuGripper6" : Bool = PLC HMI.CloseInManuGripper6 AT %DB8.DBX2.7, 100 ms
   "HMI_CloseInManuGripper7" : Bool = PLC HMI.CloseInManuGripper7 AT %DB8.DBX3.0, 100 ms
   "HMI_CloseInManuGripper8" : Bool = PLC HMI.CloseInManuGripper8 AT %DB8.DBX3.1, 100 ms
   "HMI_TableGrippersUP" : Bool = PLC HMI.TableGrippersUP AT %DB8.DBX3.2, 100 ms
   "HMI_TableGripperDown" : Bool = PLC HMI.TableGripperDown AT %DB8.DBX3.3, 100 ms
   "HMI_TablePinsUp" : Bool = PLC HMI.TablePinsUp AT %DB8.DBX3.4, 100 ms
   "HMI_TablePinsDown" : Bool = PLC HMI.TablePinsDown AT %DB8.DBX3.5, 100 ms
   "diSE_OpenGripper1" : Bool = PLC diSE_OpenGripper1 AT %I0.0, 100 ms
   "diSE_OpenGripper2" : Bool = PLC diSE_OpenGripper2 AT %I0.1, 100 ms
   "diSE_OpenGripper3" : Bool = PLC diSE_OpenGripper3 AT %I0.2, 100 ms
   "diSE_OpenGripper4" : Bool = PLC diSE_OpenGripper4 AT %I0.3, 100 ms
   "diSE_OpenGripper5" : Bool = PLC diSE_OpenGripper5 AT %I0.4, 100 ms
   "diSE_OpenGripper6" : Bool = PLC diSE_OpenGripper6 AT %I0.5, 100 ms
   "diSE_OpenGripper7" : Bool = PLC diSE_OpenGripper7 AT %I0.6, 100 ms
   "diSE_OpenGripper8" : Bool = PLC diSE_OpenGripper8 AT %I0.7, 100 ms
   "diSE_PresencePin1" : Bool = PLC diSE_PresencePin1 AT %I1.0, 100 ms
   "diSE_PresencePin2" : Bool = PLC diSE_PresencePin2 AT %I1.1, 100 ms
   "diSE_PresencePin3" : Bool = PLC diSE_PresencePin3 AT %I1.2, 100 ms
   "diSE_PresencePin4" : Bool = PLC diSE_PresencePin4 AT %I1.3, 100 ms
   "diSE_PresencePin5" : Bool = PLC diSE_PresencePin5 AT %I1.4, 100 ms
   "diSE_PresencePin6" : Bool = PLC diSE_PresencePin6 AT %I1.5, 100 ms
   "diSE_PresencePin7" : Bool = PLC diSE_PresencePin7 AT %I8.0, 100 ms
   "diSE_PresencePin8" : Bool = PLC diSE_PresencePin8 AT %I8.1, 100 ms
   "Variable_FirstScanDone" : Bool = PLC Variable.FirstScanDone AT %DB1.DBX0.0, 100 ms
   "Variable_SetMachineInitialStatus" : Bool = PLC Variable.SetMachineInitialStatus AT %DB1.DBX0.6, 100 ms
   "Variable_M_EvTableGrippres" : Bool = PLC Variable.M_EvTableGrippres AT %DB1.DBX0.7, 100 ms
   "Variable_M_EvTablePins" : Bool = PLC Variable.M_EvTablePins AT %DB1.DBX1.0, 100 ms
   "Variable_OutBuzzerPinActivatedByTube1" : Bool = PLC Variable.OutBuzzerPinActivatedByTube1 AT %DB1.DBX1.1, 100 ms
   "Variable_OutBuzzerPinActivatedByTube2" : Bool = PLC Variable.OutBuzzerPinActivatedByTube2 AT %DB1.DBX1.2, 100 ms
   "Variable_OutBuzzerPinActivatedByTube3" : Bool = PLC Variable.OutBuzzerPinActivatedByTube3 AT %DB1.DBX1.3, 100 ms
   "Variable_OutBuzzerPinActivatedByTube4" : Bool = PLC Variable.OutBuzzerPinActivatedByTube4 AT %DB1.DBX1.4, 100 ms
   "Variable_OutBuzzerPinActivatedByTube5" : Bool = PLC Variable.OutBuzzerPinActivatedByTube5 AT %DB1.DBX1.5, 100 ms
   "Variable_OutBuzzerPinActivatedByTube6" : Bool = PLC Variable.OutBuzzerPinActivatedByTube6 AT %DB1.DBX1.6, 100 ms
   "Variable_OutBuzzerPinActivatedByTube7" : Bool = PLC Variable.OutBuzzerPinActivatedByTube7 AT %DB1.DBX1.7, 100 ms
   "Variable_OutBuzzerPinActivatedByTube8" : Bool = PLC Variable.OutBuzzerPinActivatedByTube8 AT %DB1.DBX2.0, 100 ms
   "Variable_BuzzerDurationSignal" : Time = PLC Variable.BuzzerDurationSignal AT %DB1.DBD4, 100 ms
   "Variable_SignalBuzzerPinPresent" : Bool = PLC Variable.SignalBuzzerPinPresent AT %DB1.DBX8.0, 100 ms
   "Variable_M_PinsNotActivated" : Bool = PLC Variable.M_PinsNotActivated AT %DB1.DBX8.1, 100 ms
   "Variable_M_PinsActivated" : Bool = PLC Variable.M_PinsActivated AT %DB1.DBX8.2, 100 ms
   "Variable_M_GrippersOpened" : Bool = PLC Variable.M_GrippersOpened AT %DB1.DBX8.3, 100 ms
   "Variable_M_GrippersClosed" : Bool = PLC Variable.M_GrippersClosed AT %DB1.DBX8.4, 100 ms
   "Variable_M_PinsTableUpPosition" : Bool = PLC Variable.M_PinsTableUpPosition AT %DB1.DBX8.5, 100 ms
   "Variable_M_PinsTableDownPosition" : Bool = PLC Variable.M_PinsTableDownPosition AT %DB1.DBX8.6, 100 ms
   "Variable_M_GrippersTableUpPositon" : Bool = PLC Variable.M_GrippersTableUpPositon AT %DB1.DBX8.7, 100 ms
   "Variable_M_GrippersTableDownPositon" : Bool = PLC Variable.M_GrippersTableDownPositon AT %DB1.DBX9.0, 100 ms
   "Variable_M_EvGripperOutput1" : Bool = PLC Variable.M_EvGripperOutput1 AT %DB1.DBX10.1, 100 ms
   "Variable_M_EvGripperOutput2" : Bool = PLC Variable.M_EvGripperOutput2 AT %DB1.DBX10.2, 100 ms
   "Variable_M_EvGripperOutput3" : Bool = PLC Variable.M_EvGripperOutput3 AT %DB1.DBX10.3, 100 ms
   "Variable_M_EvGripperOutput4" : Bool = PLC Variable.M_EvGripperOutput4 AT %DB1.DBX10.4, 100 ms
   "Variable_M_EvGripperOutput5" : Bool = PLC Variable.M_EvGripperOutput5 AT %DB1.DBX10.5, 100 ms
   "Variable_M_EvGripperOutput6" : Bool = PLC Variable.M_EvGripperOutput6 AT %DB1.DBX10.6, 100 ms
   "Variable_M_EvGripperOutput7" : Bool = PLC Variable.M_EvGripperOutput7 AT %DB1.DBX10.7, 100 ms
   "Variable_M_EvGripperOutput8" : Bool = PLC Variable.M_EvGripperOutput8 AT %DB1.DBX11.0, 100 ms
   "Variable_M_ReadyForFirstCycle" : Bool = PLC Variable.M_ReadyForFirstCycle AT %DB1.DBX11.1, 100 ms
   "Variable_M_PreparePositionForFirstStart" : Bool = PLC Variable.M_PreparePositionForFirstStart AT %DB1.DBX11.2, 100 ms
   "Variable_M_StartCycleButtons" : Bool = PLC Variable.M_StartCycleButtons AT %DB1.DBX11.3, 100 ms
   "Variable_M_EvGrippresInitial" : Bool = PLC Variable.M_EvGrippresInitial AT %DB1.DBX11.4, 100 ms
   "Variable_M_EvTablePinsInitial" : Bool = PLC Variable.M_EvTablePinsInitial AT %DB1.DBX11.5, 100 ms
   "Variable_M_EvGripperOutputInitial" : Bool = PLC Variable.M_EvGripperOutputInitial AT %DB1.DBX11.6, 100 ms
   "Variable_M_AutomaticModePermissionToCloseGrippers" : Bool = PLC Variable.M_AutomaticModePermissionToCloseGrippers AT %DB1.DBX11.7, 100 ms
   "diSE_LeftActuatorGrippersUpPosition" : Bool = PLC diSE_LeftActuatorGrippersUpPosition AT %I8.2, 100 ms
   "diSE_LeftActuatorGrippersDownPosition" : Bool = PLC diSE_LeftActuatorGrippersDownPosition AT %I8.3, 100 ms
   "diSE_LeftActuatorTablePinsDownPosition" : Bool = PLC diSE_LeftActuatorTablePinsDownPosition AT %I8.4, 100 ms
   "diSE_LeftActuatorTablePinsUpPositon" : Bool = PLC diSE_LeftActuatorTablePinsUpPositon AT %I8.5, 100 ms
   "diSE_RightActuatorTablePinsDownPositon" : Bool = PLC diSE_RightActuatorTablePinsDownPositon AT %I8.6, 100 ms
   "diSE_RightActuatorTablePinsUpPosition" : Bool = PLC diSE_RightActuatorTablePinsUpPosition AT %I8.7, 100 ms
   "diSE_RightActuatorGripperUpPosition" : Bool = PLC diSE_RightActuatorGripperUpPosition AT %I9.0, 100 ms
   "diSE_RightActuatorGripperDownPositon" : Bool = PLC diSE_RightActuatorGripperDownPositon AT %I9.1, 100 ms
   "diPressOpenedUp" : Bool = PLC diPressOpenedUp AT %I9.4, 100 ms
   "diPressClosedDown" : Bool = PLC diPressClosedDown AT %I9.6, 100 ms
   "diPreventaOK" : Bool = PLC diPreventaOK AT %I9.2, 100 ms
   "diBT_Reset" : Bool = PLC diBT_Reset AT %I9.3, 100 ms
   "diBT_StartCycle2" : Bool = PLC diBT_StartCycle2 AT %I9.5, 100 ms
   "diPressInjectionEnd" : Bool = PLC diPressInjectionEnd AT %I9.7, 100 ms
   "dqPermitToClosePress" : Bool = PLC dqPermitToClosePress AT %Q0.0, 100 ms
   "dqPressInterface1" : Bool = PLC dqPressInterface1 AT %Q0.1, 100 ms
   "dqPressInterface2" : Bool = PLC dqPressInterface2 AT %Q0.2, 100 ms
   "dqPressInterface3" : Bool = PLC dqPressInterface3 AT %Q0.3, 100 ms
   "dqReserveQ0_4" : Bool = PLC dqReserveQ0_4 AT %Q0.4, 100 ms
   "dqReserveQ0_5" : Bool = PLC dqReserveQ0_5 AT %Q0.5, 100 ms
   "dqLED_RedFault" : Bool = PLC dqLED_RedFault AT %Q0.6, 100 ms
   "dqBuzzer" : Bool = PLC dqBuzzer AT %Q0.7, 100 ms
   "dqReserveQ1_0" : Bool = PLC dqReserveQ1_0 AT %Q1.0, 100 ms
   "dqReserveQ1_1" : Bool = PLC dqReserveQ1_1 AT %Q1.1, 100 ms
   "dqTablePinsUp" : Bool = PLC dqTablePinsUp AT %Q8.0, 100 ms
   "dqTablePinsDown" : Bool = PLC dqTablePinsDown AT %Q8.1, 100 ms
   "dqGrippresDown" : Bool = PLC dqGrippresDown AT %Q8.2, 100 ms
   "dqGrippersUp" : Bool = PLC dqGrippersUp AT %Q8.3, 100 ms
   "dqOpeningGripper1" : Bool = PLC dqOpeningGripper1 AT %Q8.4, 100 ms
   "dqClosingGripper1" : Bool = PLC dqClosingGripper1 AT %Q8.5, 100 ms
   "dqOpeningGripper2" : Bool = PLC dqOpeningGripper2 AT %Q8.6, 100 ms
   "dqClosingGripper2" : Bool = PLC dqClosingGripper2 AT %Q8.7, 100 ms
   "dqOpeningGripper3" : Bool = PLC dqOpeningGripper3 AT %Q9.0, 100 ms
   "dqClosingGripper3" : Bool = PLC dqClosingGripper3 AT %Q9.1, 100 ms
   "dqOpeningGripper4" : Bool = PLC dqOpeningGripper4 AT %Q9.2, 100 ms
   "dqClosingGripper4" : Bool = PLC dqClosingGripper4 AT %Q9.3, 100 ms
   "dqOpeningGripper5" : Bool = PLC dqOpeningGripper5 AT %Q9.4, 100 ms
   "dqClosingGripper5" : Bool = PLC dqClosingGripper5 AT %Q9.5, 100 ms
   "dqOpeningGripper6" : Bool = PLC dqOpeningGripper6 AT %Q9.6, 100 ms
   "dqClosingGripper6" : Bool = PLC dqClosingGripper6 AT %Q9.7, 100 ms
   "dqOpeningGripper7" : Bool = PLC dqOpeningGripper7 AT %Q12.0, 100 ms
   "dqClosingGripper7" : Bool = PLC dqClosingGripper7 AT %Q12.1, 100 ms
   "dqOpeningGripper8" : Bool = PLC dqOpeningGripper8 AT %Q12.2, 100 ms
   "dqClosingGripper8" : Bool = PLC dqClosingGripper8 AT %Q12.3, 100 ms
   "dqReserveq12_4" : Bool = PLC dqReserveq12_4 AT %Q12.4, 100 ms
   "dqReserveq12_5" : Bool = PLC dqReserveq12_5 AT %Q12.5, 100 ms
   "dqReserveq12_6" : Bool = PLC dqReserveq12_6 AT %Q12.6, 100 ms
   "dqReserveq12_7" : Bool = PLC dqReserveq12_7 AT %Q12.7, 100 ms
   "HMI_OpenManuAllGrippers" : Bool = PLC HMI.OpenManuAllGrippers AT %DB8.DBX3.6, 100 ms

HMI tags "AlarmsTagsHMI"
   "AlarmEvent" : Int AT %DB17.DBW0, 1 s

discrete alarms
   1: '', class Errors
   2: 'Alarm Gripper nr 4', class Errors, trigger "AlarmEvent" bit 0
   3: 'Alarm Gripper nr 5', class Errors, trigger "AlarmEvent" bit 1
   4: 'Alarm Gripper nr 6', class Errors, trigger "AlarmEvent" bit 2
   5: 'Alarm Gripper nr 7', class Errors, trigger "AlarmEvent" bit 3
   6: 'Alarm Gripper nr 8', class Errors, trigger "AlarmEvent" bit 4
   7: '', class Errors, trigger "AlarmEvent" bit 5
   8: '', class Errors, trigger "AlarmEvent" bit 6
   9: '', class Errors, trigger "AlarmEvent" bit 7
   10: 'Alarm Occured', class Errors, trigger "AlarmEvent" bit 8
   11: 'Alarm Left Actuator Grippers', class Errors, trigger "AlarmEvent" bit 9
   12: 'Alarm Right Actuator Grippers', class Errors, trigger "AlarmEvent" bit 10
   13: 'Alarm Left Actuator Pins', class Errors, trigger "AlarmEvent" bit 11
   14: 'Alarm Rihgt Actuator Pins', class Errors, trigger "AlarmEvent" bit 12
   15: 'Alarm Gripper 1', class Errors, trigger "AlarmEvent" bit 13
   16: 'Alarm Gripper 2', class Errors, trigger "AlarmEvent" bit 14
   17: 'Alarm Gripper 3', class Errors, trigger "AlarmEvent" bit 15

screen "Root screen" 480x272, template "Template_1"
   Button "Button_1" at 4,13 size 58x108; TextOff '1'
      on Press: SetBit("HMI_OpenInAutoGripper1")
      on Release: ResetBit("HMI_OpenInAutoGripper1")
      Appearance <- "diSE_PresencePin1"
   Button "Button_2" at 67,13 size 58x108; TextOff '2'
      on Release: ResetBit("HMI_OpenInAutoGripper2")
      Appearance <- "diSE_PresencePin2"
      on Press: SetBit("HMI_OpenInAutoGripper2")
   Button "Button_3" at 122,13 size 58x108; TextOff '3'
      on Press: SetBit("HMI_OpenInAutoGripper3")
      on Release: ResetBit("HMI_OpenInAutoGripper3")
      Appearance <- "diSE_PresencePin3"
   Button "Button_4" at 181,13 size 58x108; TextOff '4'
      on Release: ResetBit("HMI_OpenInAutoGripper4")
      on Press: SetBit("HMI_OpenInAutoGripper4")
      Appearance <- "diSE_PresencePin4"
   Button "Button_5" at 240,13 size 58x108; TextOff '5'
      on Press: SetBit("HMI_OpenInAutoGripper5")
      on Release: ResetBit("HMI_OpenInAutoGripper5")
      Appearance <- "diSE_PresencePin5"
   Button "Button_6" at 299,13 size 58x108; TextOff '6'
      on Press: SetBit("HMI_OpenInAutoGripper6")
      on Release: ResetBit("HMI_OpenInAutoGripper6")
      Appearance <- "diSE_PresencePin6"
   Button "Button_7" at 358,13 size 58x108; TextOff '7'
      on Press: SetBit("HMI_OpenInAutoGripper7")
      on Release: ResetBit("HMI_OpenInAutoGripper7")
      Appearance <- "diSE_PresencePin7"
   Button "Button_8" at 417,13 size 58x108; TextOff '8'
      on Press: SetBit("HMI_OpenInAutoGripper8")
      on Release: ResetBit("HMI_OpenInAutoGripper8")
      Appearance <- "diSE_PresencePin8"
   Circle "Circle_1" at 23,134 size 32x32
      Appearance <- "diPressOpenedUp"
   Circle "Circle_2" at 23,169 size 32x32
      Appearance <- "diPressClosedDown"
   Circle "Circle_3" at 23,204 size 32x32
      Appearance <- "dqPermitToClosePress"
   Circle "Circle_4" at 23,237 size 32x32
      Appearance <- "diPressInjectionEnd"
   TextField "Text field_1" at 63,141 size 93x20; Text 'MOLD OPENED'
   TextField "Text field_2" at 64,178 size 93x20; Text 'MOLD CLOSED'
   TextField "Text field_3" at 65,213 size 161x20; Text 'MOLD READY TO COLOSE'
   TextField "Text field_4" at 66,245 size 96x20; Text 'END INJECTION'
   TextField "Text field_5" at 362,212 size 94x25; Text 'F1 - HOME'
   TextField "Text field_7" at 362,232 size 115x25; Text 'F3 - ALARMS'
   Button "Button_9" at 248,134 size 96x64; TextOff 'AUTOMATIC'
      Appearance <- "HMI_Auto"
      on Press: SetBit("HMI_Auto"); ResetBit("HMI_Manu")
   Button "Button_10" at 366,134 size 96x64; TextOff 'MANUAL'
      on Press: SetBit("HMI_Manu"); ResetBit("HMI_Auto"); ActivateScreen("ManualControl", 0)
      Appearance <- "HMI_Manu"
      Visibility <- "diPressOpenedUp"

screen "Alarms" 480x272
   TextField "Text field_1" at 218,2 size 64x20; Text 'ALARMS'
   AlarmView "Alarm view_1" at 0,22 size 480x249

screen "ManualControl" 480x272
   Softkey "Softkey_F1" at 0,0 size 0x0
      on KeyDown: ActivateScreen("Root screen", 0)
   Softkey "Softkey_F2" at 0,0 size 0x0
      on KeyDown: ActivateScreen("ManualControl", 0)
   Softkey "Softkey_F3" at 0,0 size 0x0
      on KeyDown: ActivateScreen("Alarms", 0)
   TextField "Text field_1" at 174,0 size 120x20; Text 'MANUAL CONTROL'
   Button "Button_1" at 12,33 size 54x32; TextOff 'Open 1'
      on Press: SetBit("HMI_OpenInManuGripper1")
      on Release: ResetBit("HMI_OpenInManuGripper1")
      Appearance <- "diSE_OpenGripper1"
   Button "Button_2" at 12,85 size 54x32; TextOff 'Close 1'
      on Press: SetBit("HMI_CloseInManuGripper1")
      on Release: ResetBit("HMI_CloseInManuGripper1")
      Appearance <- "diSE_OpenGripper1"
   Button "Button_3" at 69,33 size 54x32; TextOff 'Open 2'
      on Press: SetBit("HMI_OpenInManuGripper2")
      on Release: ResetBit("HMI_OpenInManuGripper2")
      Appearance <- "diSE_OpenGripper2"
   Button "Button_4" at 69,85 size 54x32; TextOff 'Close 2'
      on Press: SetBit("HMI_CloseInManuGripper2")
      on Release: ResetBit("HMI_CloseInManuGripper2")
      Appearance <- "diSE_OpenGripper2"
   Button "Button_5" at 126,33 size 54x32; TextOff 'Open 3'
      on Press: SetBit("HMI_OpenInManuGripper3")
      on Release: ResetBit("HMI_OpenInManuGripper3")
      Appearance <- "diSE_OpenGripper3"
   Button "Button_6" at 126,85 size 54x32; TextOff 'Close 3'
      on Press: SetBit("HMI_CloseInManuGripper3")
      on Release: ResetBit("HMI_CloseInManuGripper3")
      Appearance <- "diSE_OpenGripper3"
   Button "Button_7" at 183,33 size 54x32; TextOff 'Open 4'
      on Press: SetBit("HMI_OpenInManuGripper4")
      on Release: ResetBit("HMI_OpenInManuGripper4")
      Appearance <- "diSE_OpenGripper4"
   Button "Button_8" at 183,85 size 54x32; TextOff 'Close 4'
      on Press: SetBit("HMI_CloseInManuGripper4")
      on Release: ResetBit("HMI_CloseInManuGripper4")
      Appearance <- "diSE_OpenGripper4"
   Button "Button_9" at 240,33 size 54x32; TextOff 'Open 5'
      on Press: SetBit("HMI_OpenInManuGripper5")
      on Release: ResetBit("HMI_OpenInManuGripper5")
      Appearance <- "diSE_OpenGripper5"
   Button "Button_10" at 240,85 size 54x32; TextOff 'Close 5'
      on Press: SetBit("HMI_CloseInManuGripper5")
      on Release: ResetBit("HMI_CloseInManuGripper5")
      Appearance <- "diSE_OpenGripper5"
   Button "Button_11" at 297,33 size 54x32; TextOff 'Open 6'
      on Press: SetBit("HMI_OpenInManuGripper6")
      on Release: ResetBit("HMI_OpenInManuGripper6")
      Appearance <- "diSE_OpenGripper6"
   Button "Button_12" at 297,85 size 54x32; TextOff 'Close 6'
      on Press: SetBit("HMI_CloseInManuGripper6")
      on Release: ResetBit("HMI_CloseInManuGripper6")
      Appearance <- "diSE_OpenGripper6"
   Button "Button_13" at 354,33 size 54x32; TextOff 'Open 7'
      on Press: SetBit("HMI_OpenInManuGripper7")
      on Release: ResetBit("HMI_OpenInManuGripper7")
      Appearance <- "diSE_OpenGripper7"
   Button "Button_14" at 354,85 size 54x32; TextOff 'Close 7'
      on Press: SetBit("HMI_CloseInManuGripper7")
      on Release: ResetBit("HMI_CloseInManuGripper7")
      Appearance <- "diSE_OpenGripper7"
   Button "Button_15" at 411,33 size 54x32; TextOff 'Open 8'
      on Press: SetBit("HMI_OpenInManuGripper8")
      on Release: ResetBit("HMI_OpenInManuGripper8")
      Appearance <- "diSE_OpenGripper8"
   Button "Button_16" at 411,85 size 54x32; TextOff 'Close 8'
      on Press: SetBit("HMI_CloseInManuGripper8")
      on Release: ResetBit("HMI_CloseInManuGripper8")
      Appearance <- "diSE_OpenGripper8"
   Button "Button_17" at 67,177 size 96x32; TextOff 'UP'
      on Press: SetBit("HMI_TablePinsUp")
      on Release: ResetBit("HMI_TablePinsUp")
      Appearance <- "Variable_M_PinsTableUpPosition"
   Button "Button_18" at 67,221 size 96x32; TextOff 'DOWN'
      on Press: SetBit("HMI_TablePinsDown")
      on Release: ResetBit("HMI_TablePinsDown")
      Appearance <- "Variable_M_PinsTableDownPosition"
   Button "Button_19" at 312,173 size 96x32; TextOff 'UP'
      on Press: SetBit("HMI_TableGrippersUP")
      on Release: ResetBit("HMI_TableGrippersUP")
      Appearance <- "Variable_M_GrippersTableUpPositon"
   Button "Button_20" at 312,215 size 96x32; TextOff 'DOWN'
      on Press: SetBit("HMI_TableGripperDown")
      on Release: ResetBit("HMI_TableGripperDown")
      Appearance <- "Variable_M_GrippersTableDownPositon"
   TextField "Text field_2" at 86,148 size 77x20; Text 'PINS TABLE'
   TextField "Text field_3" at 314,149 size 110x20; Text 'GRIPPERS TABLE'
   Button "Button_21" at 192,130 size 96x32; TextOff 'Open All'
      on Press: function_b14e0dd5("HMI_OpenManuAllGrippers", 0)
*)